// TwinCAT 3 PLC project PLC_MOTION
// Title: PLC_MOTION_LAYER
// Author: D. Hauer
// ProjectVersion: 01.00.34
// Description: MC-PtP, NCI, Camming cyclic execution layer for motion commands
// ProgramVersion: 3.1.4026.19
// libraries:
//   Tc2_EtherCAT, * (Beckhoff Automation GmbH)
//   Tc2_MC2, * (Beckhoff Automation GmbH)
//   Tc2_MC2_Camming, * (Beckhoff Automation GmbH)
//   Tc2_MC2_Drive, * (Beckhoff Automation GmbH)
//   Tc2_MC2_XFC, * (Beckhoff Automation GmbH)
//   Tc2_NCI, * (Beckhoff Automation GmbH)
//   Tc2_PlcInterpolation, * (Beckhoff Automation GmbH)
//   Tc2_Standard, * (Beckhoff Automation GmbH)
//   Tc2_System, * (Beckhoff Automation GmbH)
//   Tc2_Utilities, * (Beckhoff Automation GmbH)
//   Tc3_Module, * (Beckhoff Automation GmbH)
// project tree:
//   / CAM.TcPOU, FUNCTIONS.TcPOU, NCI.TcPOU, MAIN.TcPOU, PlcTask.TcTTO, Visualization Manager.TcVMO (not stored)
//   CAM/ FB_CamAxis.TcPOU, FB_CamCtrl.TcPOU, I_Cam_Ctrl.TcIO
//   CAM/types/ ST_CAM_CTRL.TcDUT (not stored), ST_CAM_DATA.TcDUT (not stored), ST_CAM_INFO.TcDUT (not stored), ST_CAM_READ_VALUES_PARAMETER.TcDUT, ST_CAM_STATE.TcDUT (not stored), ST_CAM_OPTIONS.TcDUT (not stored), ST_CAM_SCALING_DATA.TcDUT, ST_MOTION_FUNCTION.TcDUT (not stored), ST_MOTION_FUNCTION_POINT.TcDUT (not stored)
//   FUNCTIONS/TOUCH_PROBE/ FB_TouchProbe.TcPOU, I_TouchProbe.TcIO
//   FUNCTIONS/TOUCH_PROBE/types/ ST_2BIT.TcDUT (not stored), ST_CTRL_TOUCH_PROBE.TcDUT (not stored), ST_DC_Input.TcDUT (not stored), ST_MTI_INPUT.TcDUT (not stored), ST_MTI_STATUS.TcDUT (not stored), ST_STATE_TOUCH_PROBE.TcDUT (not stored)
//   FUNCTIONS/TRIGGER_BOX/ FB_TriggerBox.TcPOU, I_TriggerBox.TcIO
//   FUNCTIONS/TRIGGER_BOX/types/ ST_CTRL_TRIGGER.TcDUT (not stored), ST_DC_Output.TcDUT (not stored), ST_DC_State.TcDUT (not stored), ST_STATE_TRIGGER.TcDUT, T_TriggerControlBits.TcDUT
//   MAPPING/ MAPPING_in.TcPOU (not stored), MAPPING_out.TcPOU
//   MAPPING/types/ U_AXIS_CTRL.TcDUT (not stored), U_AXIS_NC_PARAMETER_WRT.TcDUT, U_AXIS_HOMING.TcDUT (not stored), U_AXIS_MOTION_OPTIONS.TcDUT, U_AXIS_MOVE_DATA.TcDUT (not stored), U_AXIS_GEAR_IN.TcDUT (not stored), U_AXIS_NC_PARAMETER_RD.TcDUT, U_AXIS_STATE.TcDUT, U_AXIS_INFO.TcDUT (not stored), U_CAM_CTRL.TcDUT, U_CAM_DATA.TcDUT (not stored), U_CAM_INFO.TcDUT (not stored), U_CAM_STATE.TcDUT (not stored), U_TOUCH_PROBE_CTRL.TcDUT (not stored), U_TOUCH_PROBE_STATE.TcDUT, U_TRIGGER_CTRL.TcDUT (not stored), U_TRIGGER_STATE.TcDUT
//   NCI/ FB_NciChannelCtrl.TcPOU (not stored), FB_NciChannel.TcPOU, I_NciChannel.TcIO (not stored), I_Nci_Ctrl.TcIO
//   NCI/types/ E_NCI_CTRL.TcDUT (not stored), E_NCI_CHANNEL_ERROR.TcDUT (not stored), E_NCI_STATE.TcDUT (not stored), E_NCI_INTERPRETER_STATE.TcDUT (not stored), ST_3D_Group.TcDUT (not stored), ST_CTRL_NCI.TcDUT (not stored), ST_NCI_M_FUNC.TcDUT (not stored), ST_Index_Group.TcDUT (not stored), ST_Interface_Group.TcDUT (not stored), ST_NciChannel_Ref.TcDUT (not stored), ST_R_Parameter.TcDUT, ST_STATE_NCI.TcDUT (not stored)
//   NC_PTP/ FB_McAxisCtrl.TcPOU, FB_McAxisBase.TcPOU, I_McAxis.TcIO (not stored)
//   NC_PTP/types/axis/ E_AxisEncoderType.TcDUT (not stored), ST_HomeParams.TcDUT (not stored)
//   NC_PTP/types/control/ E_AXIS_CTRL.TcDUT (not stored), E_AXIS_STATE.TcDUT (not stored), ST_AXIS_CTRL.TcDUT (not stored), ST_AXIS_INFO.TcDUT, ST_AXIS_STATE.TcDUT (not stored), ST_GEAR_IN.TcDUT (not stored), ST_HOMING.TcDUT (not stored), ST_MOTION_OPTIONS.TcDUT, ST_MOVE_DATA.TcDUT (not stored), ST_NC_PARAMETER.TcDUT (not stored)
//   XFC/ FB_Xfc.TcPOU
//   XFC/types/ E_XFC_CHECK.TcDUT (not stored)
//   _DUT/ E_CHECK_STATE.TcDUT (not stored), E_PROGRESS.TcDUT (not stored)
//   _GVL/ GlobalTextList.TcGTLO (not stored), GVL_AXIS.TcGVL, GVL_CAM.TcGVL (not stored), GVL_FUNCTIONS.TcGVL, GVL_MSG.TcGVL (not stored), GVL_NCI.TcGVL (not stored), PLC_CONSTANT.TcGVL (not stored), PLC_VERSION.TcGVL
//   _MSG/ fb_LocalTime.TcPOU (not stored), f_MessageSet.TcPOU, MessageData.TcPOU (not stored), T_MESSAGE_LIST.TcVIS
//   _MSG/types/ e_Device.TcDUT (not stored), E_MessageType.TcDUT (not stored), E_MESSAGE_STATE.TcDUT (not stored), e_Subdevice.TcDUT (not stored), ST_Message.TcDUT (not stored)
//   _UML/ CD_PLC_MOTION.TcCD (not stored) (excluded from build)
// real-time tasks:
//   TASK PlcTask: cycle T#10ms, priority 20, ADS port 350
//   TASK PlcTask1: cycle T#10ms, priority 21, ADS port 351
// motion (NC):
//   TASK NC-Task 1 SAF: cycle T#2ms, priority 4, ADS port 501
//   TASK NC-Task 1 SVB: cycle T#10ms, priority 8, ADS port 511
//   AXIS Axis 1 (id 1)
//     OtherSettings: AllowMotionCmdToSlave=true
//     encoder EncType=1
//     drive DrvType=5
//       Analog: TorqueSetpointScale=10, ScaleFactorActTorque=0.1
//       TimeComp: TaskDelayCycles=1
//     controller CtrType=1
//       CtrPara: PriorControlFactor=1
//         Observer: BandWidth=20
//   AXIS Axis 2 (id 2)
//     OtherSettings: AllowMotionCmdToSlave=true
//     encoder EncType=1
//     drive DrvType=5
//       Analog: TorqueSetpointScale=10, ScaleFactorActTorque=0.1
//       TimeComp: TaskDelayCycles=1
//     controller CtrType=1
//       CtrPara: PriorControlFactor=1
//         Observer: BandWidth=20
//   AXIS Axis 3 (id 3)
//     OtherSettings: AllowMotionCmdToSlave=true
//     encoder EncType=1
//     drive DrvType=5
//       Analog: TorqueSetpointScale=10, ScaleFactorActTorque=0.1
//       TimeComp: TaskDelayCycles=1
//     controller CtrType=1
//       CtrPara: PriorControlFactor=1
//         Observer: BandWidth=20
//   AXIS Axis 4 (id 4)
//     OtherSettings: AllowMotionCmdToSlave=true
//     encoder EncType=1
//     drive DrvType=5
//       Analog: TorqueSetpointScale=10, ScaleFactorActTorque=0.1
//       TimeComp: TaskDelayCycles=1
//     controller CtrType=1
//       CtrPara: PriorControlFactor=1
//         Observer: BandWidth=20
//   AXIS Axis 5 (id 5)
//     OtherSettings: AllowMotionCmdToSlave=true
//     encoder EncType=1
//     drive DrvType=5
//       Analog: TorqueSetpointScale=10, ScaleFactorActTorque=0.1
//       TimeComp: TaskDelayCycles=1
//     controller CtrType=1
//       CtrPara: PriorControlFactor=1
//         Observer: BandWidth=20
//   AXIS Axis 6 (id 6)
//     OtherSettings: AllowMotionCmdToSlave=true
//     encoder EncType=1
//     drive DrvType=5
//       Analog: TorqueSetpointScale=10, ScaleFactorActTorque=0.1
//       TimeComp: TaskDelayCycles=1
//     controller CtrType=1
//       CtrPara: PriorControlFactor=1
//         Observer: BandWidth=20
// variable links:
//   PLC_MOTION/PLC_MOTION Instance <-> NC-Task 1 SAF/Axes/Axis 1
//     PlcTask Inputs/GVL_AXIS.AxisRef[1].NcToPlc <-> Outputs/ToPlc
//     PlcTask Outputs/GVL_AXIS.AxisRef[1].PlcToNc <-> Inputs/FromPlc
//   PLC_MOTION/PLC_MOTION Instance <-> NC-Task 1 SAF/Axes/Axis 2
//     PlcTask Inputs/GVL_AXIS.AxisRef[2].NcToPlc <-> Outputs/ToPlc
//     PlcTask Outputs/GVL_AXIS.AxisRef[2].PlcToNc <-> Inputs/FromPlc
//   PLC_MOTION/PLC_MOTION Instance <-> NC-Task 1 SAF/Axes/Axis 3
//     PlcTask Inputs/GVL_AXIS.AxisRef[3].NcToPlc <-> Outputs/ToPlc
//     PlcTask Outputs/GVL_AXIS.AxisRef[3].PlcToNc <-> Inputs/FromPlc
//   PLC_MOTION/PLC_MOTION Instance <-> NC-Task 1 SAF/Axes/Axis 4
//     PlcTask Inputs/GVL_AXIS.AxisRef[4].NcToPlc <-> Outputs/ToPlc
//     PlcTask Outputs/GVL_AXIS.AxisRef[4].PlcToNc <-> Inputs/FromPlc
//   PLC_MOTION/PLC_MOTION Instance <-> NC-Task 1 SAF/Axes/Axis 5
//     PlcTask Inputs/GVL_AXIS.AxisRef[5].NcToPlc <-> Outputs/ToPlc
//     PlcTask Outputs/GVL_AXIS.AxisRef[5].PlcToNc <-> Inputs/FromPlc
//   PLC_MOTION/PLC_MOTION Instance <-> NC-Task 1 SAF/Axes/Axis 6
//     PlcTask Inputs/GVL_AXIS.AxisRef[6].NcToPlc <-> Outputs/ToPlc
//     PlcTask Outputs/GVL_AXIS.AxisRef[6].PlcToNc <-> Inputs/FromPlc

CONFIGURATION PLC_MOTION
    RESOURCE PLC ON TwinCAT3
        TASK PlcTask(INTERVAL := T#10ms, PRIORITY := 20);
        PROGRAM MAPPING_in WITH PlcTask : MAPPING_in;
        PROGRAM MAIN WITH PlcTask : MAIN;
        PROGRAM FUNCTIONS WITH PlcTask : FUNCTIONS;
        PROGRAM NCI WITH PlcTask : NCI;
        PROGRAM CAM WITH PlcTask : CAM;
        PROGRAM MAPPING_out WITH PlcTask : MAPPING_out;
    END_RESOURCE
END_CONFIGURATION

// ---- CAM/types/ST_CAM_READ_VALUES_PARAMETER.TcDUT
{attribute 'pack_mode' := '2'}
TYPE ST_CAM_READ_VALUES_PARAMETER :
STRUCT
  nValueSelectMask        : UINT;   // ReadMotionFunctionValues
  rValueMasterStart       : LREAL;  // ReadMotionFunctionValues
  rValueMasterEnd         : LREAL;  // ReadMotionFunctionValues
  rIncrement              : LREAL;
END_STRUCT
END_TYPE

// ---- CAM/types/ST_CAM_SCALING_DATA.TcDUT
{attribute 'pack_mode' := '2'}
TYPE ST_CAM_SCALING_DATA :
STRUCT
  bMasterRelative         : BIT;
  bSlaveRelative          : BIT;

  // scaling of X-axis (Master) of the CAM
  nMasterScalingMode      : UINT;
  rMasterOffset           : LREAL;
  rMasterScaling          : LREAL := 1.0;

  // scaling of Y-axis (Slave) of CAM
  nSlaveScalingMode       : UINT;

  rSlaveOffset            : LREAL;
  rSlaveScaling           : LREAL := 1.0;
END_STRUCT
END_TYPE

// ---- FUNCTIONS/TRIGGER_BOX/types/ST_STATE_TRIGGER.TcDUT
TYPE ST_STATE_TRIGGER :
STRUCT
  State           : UINT; // 0 := deactivated, 100 := BUSY, 1000 := DONE, 9000 := ERROR
  Init            : UINT;
  // FlashTimestamp  : ARRAY[1..GVL_FUNCTIONS.MAX_TRIGGER_COUNT] OF ULINT; // DC timestamp
  FlashPosition   : ARRAY[1..MAX_TRIGGER_COUNT] OF LREAL; // AxisPosition for DC timestamp
END_STRUCT
END_TYPE

// ---- FUNCTIONS/TRIGGER_BOX/types/T_TriggerControlBits.TcDUT
TYPE T_TriggerControlBits :
STRUCT
  Enable        : BIT;
  Init          : BIT;
  NoFeedback    : BIT;
{attribute 'hide'} 
  b3            : BIT;
{attribute 'hide'} 
  b4            : BIT;
{attribute 'hide'} 
  b5            : BIT;
{attribute 'hide'} 
  b6            : BIT;
{attribute 'hide'} 
  b7            : BIT;
END_STRUCT
END_TYPE

// ---- MAPPING/types/U_AXIS_NC_PARAMETER_WRT.TcDUT
TYPE U_AXIS_NC_PARAMETER_WRT :
UNION

  stCtrl              : ARRAY[1..MAX_AXIS] OF ST_NC_PARAMETER;

{IF defined (AXIS_MAP)}
  {info 'U_AXIS_NC_PARAMETER_WRT mapping activated'}
  byCtrl    AT %I*    : ARRAY[1..MAX_AXIS] OF
                        ARRAY[1..SIZEOF(ST_NC_PARAMETER)] OF BYTE;
{ELSE}
  byCtrl              : ARRAY[1..MAX_AXIS] OF
                        ARRAY[1..SIZEOF(ST_NC_PARAMETER)] OF BYTE;
{END_IF}
END_UNION
END_TYPE

// ---- MAPPING/types/U_AXIS_MOTION_OPTIONS.TcDUT
TYPE U_AXIS_MOTION_OPTIONS :
UNION

  stCtrl              : ARRAY[1..MAX_AXIS] OF ST_MOTION_OPTIONS;

{IF defined (AXIS_MAP)}
  {info 'U_AXIS_MOTION_OPTIONS mapping activated'}
  byCtrl    AT %I*    : ARRAY[1..MAX_AXIS] OF
                        ARRAY[1..SIZEOF(ST_MOTION_OPTIONS)] OF BYTE;
{ELSE}
  byCtrl              : ARRAY[1..MAX_AXIS] OF
                        ARRAY[1..SIZEOF(ST_MOTION_OPTIONS)] OF BYTE;
{END_IF}
END_UNION
END_TYPE

// ---- MAPPING/types/U_AXIS_NC_PARAMETER_RD.TcDUT
TYPE U_AXIS_NC_PARAMETER_RD :
UNION

  stState             : ARRAY[1..MAX_AXIS] OF ST_NC_PARAMETER;

{IF defined (AXIS_MAP)}
  {info 'U_AXIS_NC_PARAMETER_RD mapping activated'}
  byState   AT %Q*    : ARRAY[1..MAX_AXIS] OF
                        ARRAY[1..SIZEOF(ST_NC_PARAMETER)] OF BYTE;
{ELSE}
  byState             : ARRAY[1..MAX_AXIS] OF
                        ARRAY[1..SIZEOF(ST_NC_PARAMETER)] OF BYTE;
{END_IF}
END_UNION
END_TYPE

// ---- MAPPING/types/U_AXIS_STATE.TcDUT
TYPE U_AXIS_STATE :
UNION

  stState             : ARRAY[1..MAX_AXIS] OF ST_AXIS_STATE;

{IF defined (AXIS_MAP)}
  {info 'U_AXIS_STATE mapping activated'}
  byState   AT %Q*    : ARRAY[1..MAX_AXIS] OF
                        ARRAY[1..SIZEOF(ST_AXIS_STATE)] OF BYTE;
{ELSE}
  byState             : ARRAY[1..MAX_AXIS] OF
                        ARRAY[1..SIZEOF(ST_AXIS_STATE)] OF BYTE;
{END_IF}
END_UNION
END_TYPE

// ---- MAPPING/types/U_CAM_CTRL.TcDUT
TYPE U_CAM_CTRL :
UNION
  stCtrl              : ARRAY[1..MAX_AXIS] OF ST_CAM_CTRL;

{IF defined (CAM_MAP)}
  {info 'U_CAM_CTRL mapping activated'}
  byCtrl    AT %I*    : ARRAY[1..MAX_AXIS] OF
                        ARRAY[1..SIZEOF(ST_CAM_CTRL)] OF BYTE;
{ELSE}
  byCtrl              : ARRAY[1..MAX_AXIS] OF
                        ARRAY[1..SIZEOF(ST_CAM_CTRL)] OF BYTE;
{END_IF}
END_UNION
END_TYPE

// ---- MAPPING/types/U_TOUCH_PROBE_STATE.TcDUT
TYPE U_TOUCH_PROBE_STATE :
UNION
  stState              : ARRAY[1..MAX_TOUCH_PROBE] OF ST_STATE_TOUCH_PROBE;

{IF defined (TRIGGER_MAP)}
  {info 'U_TOUCH_PROBE_STATE mapping activated'}
  byState    AT %Q*   : ARRAY[1..MAX_TOUCH_PROBE] OF
                        ARRAY[1..SIZEOF(ST_STATE_TOUCH_PROBE)] OF BYTE;
{ELSE}
  byState             : ARRAY[1..MAX_TOUCH_PROBE] OF
                        ARRAY[1..SIZEOF(ST_STATE_TOUCH_PROBE)] OF BYTE;
{END_IF}
END_UNION
END_TYPE

// ---- MAPPING/types/U_TRIGGER_STATE.TcDUT
TYPE U_TRIGGER_STATE :
UNION
  stState              : ARRAY[1..MAX_TRIGGER_BOX] OF ST_STATE_TRIGGER;

{IF defined (TRIGGER_MAP)}
  {info 'U_TRIGGER_STATE mapping activated'}
  byState    AT %Q*   : ARRAY[1..MAX_TRIGGER_BOX] OF
                        ARRAY[1..SIZEOF(ST_STATE_TRIGGER)] OF BYTE;
{ELSE}
  byState             : ARRAY[1..MAX_TRIGGER_BOX] OF
                        ARRAY[1..SIZEOF(ST_STATE_TRIGGER)] OF BYTE;
{END_IF}
END_UNION
END_TYPE

// ---- NCI/types/ST_R_Parameter.TcDUT
{attribute 'pack_mode' := '2'}
TYPE ST_R_Parameter :
STRUCT
  _nStart               : DINT := 901;
  _nCount               : DINT :=   4;
  _rValue               : ARRAY[0..MAX_R_PARA] OF LREAL;
END_STRUCT
END_TYPE

// ---- NC_PTP/types/control/ST_AXIS_INFO.TcDUT
{attribute 'pack_mode' := '2'}
TYPE ST_AXIS_INFO :
STRUCT
  bEnabled    : BIT; // Enabled: check if ControlLoop is closed and active
  bReferenced : BIT; // Axis homing bit
  bReady      : BIT; // enabled & NOT bError & no Axis Function requested
  bBusy       : BIT; // axis function requested or active
  bError      : BIT;
  bTimeout    : BIT; // for move cmds or switching drive on timeout
  bInTarget   : BIT; // ActPos = SetPos --> position check is done with configured window in NC
  bStandstill : BIT; // No Error and NOT moving
 
  nErrorId            : UDINT;

  rActPos             : LREAL;
  rActVelo            : LREAL;
  rPosDiff            : LREAL;

  dwCoupleState       : DWORD;   // cyclic information about axis couple state
  nNcAxisId           : UDINT;
END_STRUCT
END_TYPE

// ---- NC_PTP/types/control/ST_MOTION_OPTIONS.TcDUT
{attribute 'pack_mode' := '2'}
TYPE ST_MOTION_OPTIONS :
STRUCT
  eBufferMode   : Tc2_MC2.MC_BufferMode;  // used in FB_McAxisCtrl.MoverBufferPos, MoveBufferVelo
  rDistance     : LREAL;                  // used in FB_McAxis.SendToPos; axis has to move rDistance for method to be done
END_STRUCT
END_TYPE

// ---- _GVL/GVL_AXIS.TcGVL
{attribute 'qualified_only'}
VAR_GLOBAL

  // TwinCAT NC mapping cyclic reference
  //  - link to NC/PtP
  //  - a motion Ctrl function block gets REFERENCE TO all axis
  AxisRef                     : ARRAY[1..PLC_CONSTANT.MAX_AXIS] OF Tc2_MC2.AXIS_REF;

  //-----------------------------------------------------------------------------
  // interfaces of I_McAxis 
  //  - to provide access to basic MC functions in 
  //    - NCI(PRG)() / FB_NciChannelCtrl,
  //    - CAM(PRG)() / FB_CamCtrl
  //-----------------------------------------------------------------------------
  ItfMcAxis                   : ARRAY[1..PLC_CONSTANT.MAX_AXIS] OF I_McAxis;     // interface to basic MC functions


  //-----------------------------------------------------------------------------
  // command and state structure
  //  - datafields for anyone to access
  //    - ADS via symbol
  //    - cyclic mapping to any other cyclic network/runtime
  //-----------------------------------------------------------------------------
  Ctrl                        : ARRAY[1..PLC_CONSTANT.MAX_AXIS] OF ST_AXIS_CTRL;      // command structure to write into
  State                       : ARRAY[1..PLC_CONSTANT.MAX_AXIS] OF ST_AXIS_STATE;     // state structure to read from

  //-----------------------------------------------------------------------------
  // data and info structure
  //  - parameter data fields for
  //    - Ctrl  --> Data
  //    - State --> Info
  //-----------------------------------------------------------------------------
  Info                        : ARRAY[1..PLC_CONSTANT.MAX_AXIS] OF ST_AXIS_INFO;      // axis state and position data to read from
  Data                        : ARRAY[1..PLC_CONSTANT.MAX_AXIS] OF ST_MOVE_DATA;      // axis data to write into


  //-----------------------------------------------------------------------------
  // special function parameter structs
  // - additional details for axis command
  //-----------------------------------------------------------------------------
  NcParameterWrt              : ARRAY[1..PLC_CONSTANT.MAX_AXIS] OF ST_NC_PARAMETER;   // struct for a single parameter value put/get your data here before/after using Ctrl
  NcParameterRd               : ARRAY[1..PLC_CONSTANT.MAX_AXIS] OF ST_NC_PARAMETER;   // struct for a single parameter value put/get your data here before/after using Ctrl

  HomeParameter               : ARRAY[1..PLC_CONSTANT.MAX_AXIS] OF ST_HOMING;         // homing parameter for each axis

  GearInParameter             : ARRAY[1..PLC_CONSTANT.MAX_AXIS] OF ST_GEAR_IN;        // GearIn and GearInMultiMaster, index to master axes[1-4], rGearRatio[1-4]

  MotionOptions               : ARRAY[1..PLC_CONSTANT.MAX_AXIS] OF ST_MOTION_OPTIONS; // additional motion parameters


  //-----------------------------------------------------------------------------
  // cyclic interface function block: FB_McAxisCtrl
  //  - PtP MC functions are here
  //  - implements I_McAxis
  //-----------------------------------------------------------------------------
  Control                     : ARRAY[1..PLC_CONSTANT.MAX_AXIS] OF FB_McAxisCtrl;     // cyclic interface for accepting and executing orders

END_VAR

// ---- _GVL/GVL_FUNCTIONS.TcGVL
{attribute 'qualified_only'}
VAR_GLOBAL
  //-----------------------------------------------------------------------------------------------------------
  // TriggerBox for moving axis, set output to activate camera, get input timestamp from flash controller
  //-----------------------------------------------------------------------------------------------------------
{IF defined (XFC)}
  TriggerBoxCtrl                : ARRAY[1..MAX_TRIGGER_BOX] OF Fb_TriggerBox;   // execution of trigger function
{ELSE}
  TriggerBoxCtrl                : ARRAY[1..MAX_TRIGGER_BOX] OF I_TriggerBox;   // execution of trigger function
{END_IF}

  CtrlTrigger                   : ARRAY[1..MAX_TRIGGER_BOX] OF ST_CTRL_TRIGGER;
  StateTrigger                  : ARRAY[1..MAX_TRIGGER_BOX] OF ST_STATE_TRIGGER;

  DigitalOutPutDCState  AT %I*  : ARRAY[1..MAX_TRIGGER_BOX] OF ST_DC_State;

  DigitalOutputDC   AT %Q*      : ARRAY[1..MAX_TRIGGER_BOX] OF ST_DC_Output;
  DigitalInputDC    AT %I*      : ARRAY[1..MAX_TRIGGER_BOX] OF ST_DC_Input; // distributed clock digital input with timestamps positive & negative


  //-----------------------------------------------------------------------------------------------------------
  // Touch Probe with moving axis, get input timestamp within axis window, get prcise position using the timestamp
  //-----------------------------------------------------------------------------------------------------------
{IF defined (XFC)}
  TouchProbeCtrl                : ARRAY[1..MAX_TOUCH_PROBE] OF Fb_TouchProbe;   // execution of Touch probe function
{ELSE}
  TouchProbeCtrl                : ARRAY[1..MAX_TOUCH_PROBE] OF I_TouchProbe;   // execution of Touch probe function
{END_IF}

  CtrlTouchProbe                : ARRAY[1..MAX_TOUCH_PROBE] OF ST_CTRL_TOUCH_PROBE;
  StateTouchProbe               : ARRAY[1..MAX_TOUCH_PROBE] OF ST_STATE_TOUCH_PROBE;

  //DigitalInputDC    AT %I*      : ARRAY[1..MAX_TOUCH_PROBE] OF ST_DC_Input; // distributed clock digital input with timestamps positive & negative
  DigitalInput      AT %I*      : ARRAY[1..MAX_TOUCH_PROBE] OF ST_MTI_INPUT;    // multi time stamp, one channel
  DigitalState      AT %I*      : ARRAY[1..MAX_TOUCH_PROBE] OF ST_MTI_STATUS;   // multi time stamp status from terminal

END_VAR

// ---- _GVL/PLC_VERSION.TcGVL
{attribute 'qualified_only'}
VAR_GLOBAL CONSTANT
  VERSION               : STRING := 'V 01.00.34';

  // 2025 10 24 HAUD
  //
  // documentation added, 
  // project dev changed to 4026.19
  // Ambiguities resoved

  // 2025 08 21 HAUD
  //
  // e_Device: Application added
  // e_Subdevices: merge with XTS_TRANSPORT_LAYER
  // FB_McAxis: testing SendToPos, distance added to method interface

  // 2025 02 17 HAUD
  //
  // code review
  // Message Levels are set during initialization
  // sizeof mapping data is fetched at startup only

  // 2025 01 09 HAUD
  //
  // - FUNCTIONS
  //    - code review
  //    - ctrl/state mechanic harmonized
  // - MAPPING
  //    - UNIONS added

  // 2024 08 08 HAUD
  //
  // - TC_PLC_MOTION_LAYER: 
  //    - XFC base class added
  //    - TriggerBox (DC output set, DC Input latch)
  //    - TouchProbe (DC Input latch: positive, negative)

  // 2024 06 21 HAUD
  //
  // - TC_PLC_MOTION_LAYER: 
  //    - E_PROGRESS refactoring to match TC_XTS_TRANSPORT_LAYER
  

  // 2024 06 10 HAUD
  //
  // - TC_PLC_MOTION_LAYER: 
  //    - rename repository
  //    - remove LEGACY compatibility
  //
  // - PLC_OPEN_DRIVE:
  //    - deprecated


  // 2024 05 31 HAUD
  // 
  // V 01.00.02
  // precompiler defines: 
  //  - BSD: 
  //    - Tc-BSD file system is used else Windows file system is used
  //
  //  - TEST:
  //    - GVL_MSG.MessageLevel
  // Axis, Cam, Nci have individual message levels now

  // 2024 03 09 HAUD
  // 
  // V 01.00.01
  // MC PtP - execution layer with optional mapping
  // NCI    - execution layer with optional mapping
  // CAM    . execution layer with optional mapping
  // precompiler defines: 
  //  - WIN: windows file system is used else Tc-BSD file system is used
  //  - NCI: NCI libraries are linked in project
  //  - CAM: Camming libraries are linked in project
  //  - AXIS_MAP: mapping is used


  // 2024 02 15 HAUD
  // 
  // V 00.50.04
  //
  // Buffered moves test
  // CamIn Test --> TODO MultiCam
  // Message system, cyclic check for write
  

  // 2024 01 12 HAUD
  //
  // V 00.50.03
  //
  // Building is done
  // start of UnitTesting

  // 2024 01 17 HAUD
  //
  // V 00.50.02
  // 
  // start camming implementation (MC_CamIn_V2)
  // legacy namespace available for downward compatibility of ADS Symbol names

  // 2023 12 23 HAUD
  // NC_PTP
  // - redesign for PLC_OPEN_DRIVE started 
  //    --> E_PROGRESS for state feedback
  // - FB_AxisControl inherits FB_McAxis


  //  2023 10 19
  //  HAUD
  // first draft 
  // TODO: everything

END_VAR

// ---- CAM/I_Cam_Ctrl.TcIO
INTERFACE I_Cam_Ctrl

PROPERTY Axes : reference TO ARRAY[1..PLC_CONSTANT.MAX_AXIS] OF AXIS_REF
SET
END_SET
END_PROPERTY

PROPERTY AxisCtrl : pointer to ARRAY[1..PLC_CONSTANT.MAX_AXIS] OF st_axis_ctrl
SET
END_SET
END_PROPERTY

PROPERTY AxisData : pointer to ARRAY[1..PLC_CONSTANT.MAX_AXIS] OF ST_CAM_DATA
SET
END_SET
END_PROPERTY

PROPERTY AxisIndex : uint
SET
END_SET
END_PROPERTY

PROPERTY AxisInfo : pointer to ARRAY[1..PLC_CONSTANT.MAX_AXIS] OF ST_AXIS_INFO
SET
END_SET
END_PROPERTY

PROPERTY AxisState : pointer to ARRAY[1..PLC_CONSTANT.MAX_AXIS] OF ST_CAM_STATE
SET
END_SET
END_PROPERTY

METHOD Cycle  : e_progress
END_METHOD

PROPERTY ItfMcAxes : array[1..MAX_AXIS] of I_McAxis
SET
END_SET
END_PROPERTY

PROPERTY MessageLevel : E_MessageType
SET
END_SET
END_PROPERTY

PROPERTY MotionFunction : POINTER TO ARRAY[1..MAX_AXIS] OF ST_MOTION_FUNCTION
SET
END_SET
END_PROPERTY

PROPERTY MotionFunctionPoint : pointer to array[1..MAX_AXIS] of ST_MOTION_FUNCTION_POINT
SET
END_SET
END_PROPERTY

END_INTERFACE

// ---- FUNCTIONS/TOUCH_PROBE/I_TouchProbe.TcIO
INTERFACE I_TouchProbe

PROPERTY Ctrl : REFERENCE TO ARRAY [1..MAX_TOUCH_PROBE] OF ST_CTRL_TOUCH_PROBE
SET
END_SET
END_PROPERTY

METHOD Cycle : BOOL
VAR_INPUT
END_VAR
END_METHOD

PROPERTY Index : udint
GET
END_GET
SET
END_SET
END_PROPERTY

PROPERTY Input : pointer TO ARRAY [1..MAX_TOUCH_PROBE] OF ST_MTI_Input
SET
END_SET
END_PROPERTY

PROPERTY InputState : pointer TO ARRAY [1..MAX_TOUCH_PROBE] OF ST_MTI_STATUS
SET
END_SET
END_PROPERTY

PROPERTY ItfAxis : ARRAY[1..MAX_AXIS]       OF I_McAxis
SET
END_SET
END_PROPERTY

PROPERTY MessageLevel : e_messagetype
GET
END_GET
SET
END_SET
END_PROPERTY

PROPERTY State :  REFERENCE TO ARRAY[1..MAX_TOUCH_PROBE] OF ST_STATE_TOUCH_PROBE;
SET
END_SET
END_PROPERTY

END_INTERFACE

// ---- FUNCTIONS/TRIGGER_BOX/I_TriggerBox.TcIO
INTERFACE I_TriggerBox

PROPERTY Ctrl : REFERENCE TO ARRAY [1..MAX_TRIGGER_BOX] OF ST_CTRL_TRIGGER
SET
END_SET
END_PROPERTY

METHOD Cycle : BOOL
VAR_INPUT
END_VAR
END_METHOD

METHOD CycleWaitForPosition : BOOL
VAR_INPUT
END_VAR
END_METHOD

PROPERTY Index : udint
GET
END_GET
SET
END_SET
END_PROPERTY

PROPERTY Input : pointer TO ARRAY [1..MAX_TRIGGER_BOX] OF ST_DC_Input
SET
END_SET
END_PROPERTY

PROPERTY ItfAxis : ARRAY[1..MAX_AXIS]       OF I_McAxis
SET
END_SET
END_PROPERTY

PROPERTY MessageLevel : e_messagetype
GET
END_GET
SET
END_SET
END_PROPERTY

PROPERTY Output_2252 : pointer TO ARRAY [1..MAX_TRIGGER_BOX] OF ST_DC_Output
SET
END_SET
END_PROPERTY

PROPERTY State : REFERENCE TO ARRAY[1..MAX_TRIGGER_BOX] OF ST_STATE_TRIGGER
SET
END_SET
END_PROPERTY

END_INTERFACE

// ---- NCI/I_Nci_Ctrl.TcIO
INTERFACE I_Nci_Ctrl

PROPERTY ChnCtrl : pointer to ST_CTRL_NCI
SET
END_SET
END_PROPERTY

PROPERTY ChnId : udint
GET
END_GET
END_PROPERTY

PROPERTY ChnState : pointer to ST_STATE_NCI
SET
END_SET
END_PROPERTY

METHOD Cycle : E_PROGRESS
VAR_INPUT
END_VAR
END_METHOD

PROPERTY ItfChannel : I_NciChannel
GET
END_GET
END_PROPERTY

PROPERTY M_FunctionScope : pointer to st_nci_m_func
SET
END_SET
END_PROPERTY

END_INTERFACE

// ---- MAIN.TcPOU
PROGRAM MAIN
VAR
  bInit                     : BOOL;         // shall be checked by controlling entity, before using Ctrl/State structs
  eInit                     : E_PROGRESS;   // shall be checked by controlling entity, before using Ctrl/State structs

  nAxis,
  nAxisInit                 : UINT;

  stMsg                     : ST_Message;

  bWriteTimerActive         : Bool;         // you decide whether to use timed logging into file or not
  tWriteLog                 : TIME := T#10S;
  tonWriteLog               : Tc2_Standard.TON;
END_VAR


(*
//-----------------------------------------------------------------------------------------------------------------
//-----------------------------------------------------------------------------------------------------------------
// react to operation modes (how to do it in an easy self documenting way)
//-----------------------------------------------------------------------------------------------------------------
//-----------------------------------------------------------------------------------------------------------------
CASE (GVL_AXIS.State[i].eState MOD E_PROGRESS.PROGRESS_DONE)
OF
  E_AXIS_STATE.AXIS_INIT:
    ;// do something after success  

  E_AXIS_STATE.AXIS_MOVE_POS::
    ;// do something after success
ELSE
  CASE (GVL_AXIS.State[i].eState MOD E_PROGRESS.PROGRESS_ERROR)
  OF
    E_AXIS_STATE.AXIS_INIT:
      ;// do something after success  
  
    E_AXIS_STATE.AXIS_MOVE_POS::
      ;// do something after success
  ELSE
    ;// down the rabbit hole you go from here
  END_CASE
END_CASE
*)



//-----------------------------------------------------------------------------------------------------------------
// Local time; used for timestamps
//-----------------------------------------------------------------------------------------------------------------
GVL_MSG.fbLocalTime(
                    sLocalTime                => GVL_MSG.sLocalTime, 
                    dtLocalTime               => GVL_MSG.dtLocalTime);
//-----------------------------------------------------------------------------------------------------------------
//-----------------------------------------------------------------------------------------------------------------
// /assign dataflow
//-----------------------------------------------------------------------------------------------------------------
FOR nAxis := 1 TO PLC_CONSTANT.MAX_AXIS
DO
  GVL_AXIS.Control[nAxis].AxisIndex           := nAxis;

  GVL_AXIS.Control[nAxis].AxisCtrl            := ADR(GVL_AXIS.Ctrl);          // command
  GVL_AXIS.Control[nAxis].AxisState           := ADR(GVL_AXIS.State);         // state + result of command

  GVL_AXIS.Control[nAxis].Axes                REF=   GVL_AXIS.AxisRef;        // All for one; coupling requires access across all axes

  GVL_AXIS.Control[nAxis].AxisInfo            := ADR(GVL_AXIS.Info);          // axis information: act/set values and bits from axis
  GVL_AXIS.Control[nAxis].AxisData            := ADR(GVL_AXIS.Data);          // position and dynamic constraints for movement
  GVL_AXIS.Control[nAxis].AxisGearInParameter := ADR(GVL_AXIS.GearInParameter);

  GVL_AXIS.Control[nAxis].WriteNcParameter    := ADR(GVL_AXIS.NcParameterWrt);
  GVL_AXIS.Control[nAxis].ReadNcParameter     := ADR(GVL_AXIS.NcParameterRd);

  GVL_AXIS.Control[nAxis].HomingParameter     := ADR(GVL_AXIS.HomeParameter);
  GVL_AXIS.Control[nAxis].MotionOptions       := ADR(GVL_AXIS.MotionOptions);

  GVL_AXIS.ItfMcAxis[nAxis]                   := GVL_AXIS.Control[nAxis]; 
END_FOR
//-----------------------------------------------------------------------------------------------------------------
// assign dataflow/
//-----------------------------------------------------------------------------------------------------------------
//-----------------------------------------------------------------------------------------------------------------
// /INIT
// - successful init is required for other optional members to start
//-----------------------------------------------------------------------------------------------------------------
IF NOT bInit
THEN
  CASE eInit
  OF
    E_PROGRESS.PROGRESS_INVALID,
    E_PROGRESS.PROGRESS_DONE:
      FOR nAxis := 1 TO PLC_CONSTANT.MAX_AXIS
      DO
        GVL_AXIS.Control[nAxis].MessageLevel  := GVL_MSG.MessageLevelAxisPtp;
      END_FOR
      nAxisInit                               := 1;
      eInit                                   := E_PROGRESS.PROGRESS_INIT;


    E_PROGRESS.PROGRESS_INIT:
      stMsg.eType                             := E_MessageType.eMessageVerbose;
      stMsg.eDevice                           := e_Device.General;
      stMsg.eSubdevice                        := e_SubDevice.AxisStartUp;
      stMsg.iErrorNumber                      := nAxisInit;

      stMsg.sText                             := concat('MAIN.eInit: ', TO_STRING(eInit));

      IF (GVL_MSG.MessageLevelAxisPtp = E_MessageType.eMessageVerbose)
      THEN
        f_MessageSet(stMsg);
      END_IF

      GVL_AXIS.Ctrl[nAxisInit].eCmd           := E_AXIS_CTRL.AXIS_NULL;
      eInit                                   := E_PROGRESS.PROGRESS_BUSY;


    E_PROGRESS.PROGRESS_BUSY:
      GVL_AXIS.Ctrl[nAxisInit].eCmd          := E_AXIS_CTRL.AXIS_INIT;

      IF    (GVL_AXIS.State[nAxisInit].eState = E_AXIS_STATE.AXIS_INIT + E_PROGRESS.PROGRESS_ERROR)
      THEN
        eInit                                 := E_PROGRESS.PROGRESS_ERROR;

        stMsg.eType                           := E_MessageType.eMessageError;
        stMsg.eDevice                         := e_Device.General;
        stMsg.eSubdevice                      := e_SubDevice.AxisStartUp;
        stMsg.iErrorNumber                    := GVL_AXIS.Control[nAxisInit].ErrorId;

        stMsg.sText                           := concat('MAIN.eInit ERROR at Index: ', TO_STRING(nAxisInit));
        f_MessageSet(stMsg);

      ELSIF (GVL_AXIS.State[nAxisInit].eState = E_AXIS_STATE.AXIS_INIT + E_PROGRESS.PROGRESS_DONE)
      THEN
        eInit                                 := E_PROGRESS.PROGRESS_CHECK;
      END_IF


    E_PROGRESS.PROGRESS_CHECK:
      IF NOT (nAxisInit > PLC_CONSTANT.MAX_AXIS-1)
      THEN
        nAxisInit                             := nAxisInit + 1;
        eInit                                 := E_PROGRESS.PROGRESS_INIT;

      ELSE
        bInit                                 := TRUE;
        eInit                                 := E_PROGRESS.PROGRESS_DONE;

        stMsg.eType                           := E_MessageType.eMessageInfo;
        stMsg.eDevice                         := e_Device.General;
        stMsg.eSubdevice                      := e_SubDevice.AxisStartUp;
        stMsg.iErrorNumber                    := MAX_AXIS;

        stMsg.sText                           := concat('MAIN.eInit: ', TO_STRING(eInit));
        f_MessageSet(stMsg);
      END_IF
  END_CASE
END_IF
//-----------------------------------------------------------------------------------------------------------------
// INIT
//-----------------------------------------------------------------------------------------------------------------
//-----------------------------------------------------------------------------------------------------------------
// /cyclic
//-----------------------------------------------------------------------------------------------------------------
IF (eInit <> E_PROGRESS.PROGRESS_ERROR)
THEN
  FOR nAxis := 1 TO PLC_CONSTANT.MAX_AXIS
  DO
      GVL_AXIS.Control[nAxis]();
  END_FOR
END_IF
//-----------------------------------------------------------------------------------------------------------------
// cyclic/
//-----------------------------------------------------------------------------------------------------------------


//-----------------------------------------------------------------------------------------------------------------
// /logging
//-----------------------------------------------------------------------------------------------------------------
tonWriteLog(IN:= TRUE, PT := tWriteLog);

IF (tonWriteLog.Q)
THEN
  MessageData.bWriteFile      := bWriteTimerActive; // you have to decide whether to use timed write or not
  tonWriteLog(IN:= FALSE);
END_IF

//-----------------------------------------------------------------------------------------------------------------
// write message list to file
//-----------------------------------------------------------------------------------------------------------------
MessageData(pList			        := ADR(GVL_MSG.Messages),
			      pLocalTime        := ADR(GVL_MSG.dtLocalTime), 
			      bBusy=> );

// clear write trigger
IF MessageData.bWriteFile AND
   MessageData.bBusy
THEN
  MessageData.bWriteFile      := FALSE;
END_IF
//-----------------------------------------------------------------------------------------------------------------
// logging/
//-----------------------------------------------------------------------------------------------------------------

END_PROGRAM

// ---- _MSG/f_MessageSet.TcPOU
FUNCTION f_MessageSet : BOOL
VAR_INPUT
  stMessage   : ST_Message;
END_VAR
VAR
  _uiIndex   : uINT;
END_VAR

stMessage.tTime                     := GVL_MSG.sLocalTime;

FOR _uiIndex := 1 TO GVL_MSG.MAX_MESSAGE
DO
  IF (GVL_MSG.Messages[_uiIndex].eType = e_MessageType.eMessageEmpty)
  THEN
    GVL_MSG.Messages[_uiIndex]      := stMessage;
    GVL_MSG.MessageIndex            := _uiIndex;
    EXIT;
  END_IF
END_FOR

IF (stMessage.eType = E_MessageType.eMessageError)
THEN
  // in case of error: increment counter
  GVL_MSG.MessageError := GVL_MSG.MessageError + 1;
END_IF

END_FUNCTION

// ---- FUNCTIONS.TcPOU
PROGRAM FUNCTIONS
VAR
  eInit             : E_PROGRESS;

  nAxis,
  nTrigger,
  nProbe            : UINT;
END_VAR

//-----------------------------------------------------------------------------------------------------------------
// check if compiler define is present [PLC_STATE_DRIVE/CompilerDefines/Manual: XFC]
// see PLC_CONSTANT for conditional pragma
//-----------------------------------------------------------------------------------------------------------------
IF NOT PLC_CONSTANT.XFC_ACTIVE THEN eInit := E_PROGRESS.PROGRESS_NOT_EXIST; RETURN; END_IF
//-----------------------------------------------------------------------------------------------------------------
//-----------------------------------------------------------------------------------------------------------------
// check MAIN.eInit
//-----------------------------------------------------------------------------------------------------------------
IF NOT (MAIN.eInit = E_PROGRESS.PROGRESS_DONE) 
THEN
  // wait for MAIN to be fully initialized
  eInit                                               := E_PROGRESS.PROGRESS_INVALID; 
  RETURN; 
ELSE
  // at the moment FUNCTIONS does not require a general init procedure
  eInit                                               := E_PROGRESS.PROGRESS_DONE;    // general init done
END_IF
//-----------------------------------------------------------------------------------------------------------------
//-----------------------------------------------------------------------------------------------------------------
// /cyclic
//-----------------------------------------------------------------------------------------------------------------
FOR nProbe := 1 TO MAX_TOUCH_PROBE
DO
  GVL_FUNCTIONS.TouchProbeCtrl[nProbe].MessageLevel   := GVL_MSG.MessageLevelTouchProbe[nProbe];
  GVL_FUNCTIONS.TouchProbeCtrl[nProbe].Index          := nProbe;
  GVL_FUNCTIONS.TouchProbeCtrl[nProbe].ItfAxis        := GVL_AXIS.ItfMcAxis;

  GVL_FUNCTIONS.TouchProbeCtrl[nProbe].Ctrl           REF= GVL_FUNCTIONS.CtrlTouchProbe;
  GVL_FUNCTIONS.TouchProbeCtrl[nProbe].State          REF= GVL_FUNCTIONS.StateTouchProbe;

  GVL_FUNCTIONS.TouchProbeCtrl[nProbe].Input          := ADR(GVL_FUNCTIONS.DigitalInput);
  GVL_FUNCTIONS.TouchProbeCtrl[nProbe].InputState     := ADR(GVL_FUNCTIONS.DigitalState);
  GVL_FUNCTIONS.TouchProbeCtrl[nProbe].Cycle();

END_FOR

FOR nTrigger := 1 TO MAX_TRIGGER_BOX
DO
  GVL_FUNCTIONS.TriggerBoxCtrl[nTrigger].MessageLevel := GVL_MSG.MessageLevelTriggerBox[nTrigger];
  GVL_FUNCTIONS.TriggerBoxCtrl[nTrigger].Index        := nTrigger;
  GVL_FUNCTIONS.TriggerBoxCtrl[nTrigger].ItfAxis      := GVL_AXIS.ItfMcAxis;

  GVL_FUNCTIONS.TriggerBoxCtrl[nTrigger].Ctrl         REF= GVL_FUNCTIONS.CtrlTrigger;
  GVL_FUNCTIONS.TriggerBoxCtrl[nTrigger].State        REF= GVL_FUNCTIONS.StateTrigger;

  GVL_FUNCTIONS.TriggerBoxCtrl[nTrigger].Input        := ADR(GVL_FUNCTIONS.DigitalInputDC);
  GVL_FUNCTIONS.TriggerBoxCtrl[nTrigger].Output_2252  := ADR(GVL_FUNCTIONS.DigitalOutputDC);

  GVL_FUNCTIONS.TriggerBoxCtrl[nTrigger].Cycle();
END_FOR
//-----------------------------------------------------------------------------------------------------------------
// cyclic/
//-----------------------------------------------------------------------------------------------------------------
//-----------------------------------------------------------------------------------------------------------------

END_PROGRAM

// ---- NCI.TcPOU
PROGRAM NCI
VAR
  bInit                     : BOOL;
  eInit                     : E_PROGRESS;

  nChn,
  nChnInit,
  nAxis,
  nAxisInit                 : UINT;

  stMsg                     : ST_Message;

END_VAR

//-----------------------------------------------------------------------------------------------------------------
// check if compiler define is present [PLC_STATE_DRIVE/CompilerDefines/Manual: NCI]
// see PLC_CONSTANT for conditional pragma
//-----------------------------------------------------------------------------------------------------------------
IF NOT PLC_CONSTANT.NCI_ACTIVE THEN eInit   := E_PROGRESS.PROGRESS_NOT_EXIST; RETURN; END_IF
//-----------------------------------------------------------------------------------------------------------------
//-----------------------------------------------------------------------------------------------------------------
// check for MAIN.eInit
//-----------------------------------------------------------------------------------------------------------------
IF NOT (MAIN.eInit = E_PROGRESS.PROGRESS_DONE) THEN eInit   := E_PROGRESS.PROGRESS_INVALID; RETURN; END_IF
//-----------------------------------------------------------------------------------------------------------------
//-----------------------------------------------------------------------------------------------------------------
// /assign dataflow
//-----------------------------------------------------------------------------------------------------------------
FOR nChn := 1 TO MAX_NCI_CH
DO
  // NCI axis configuration --> NC AxisId used
  GVL_NCI.fbNciCtrl[nChn].ItfChannel.CfgAxes          := ADR(GVL_NCI.stAxisConfig[nChn]);

  // R Parameter properties
  GVL_NCI.fbNciCtrl[nChn].ItfChannel.R_ParameterRead  := ADR(GVL_NCI.R_ParameterRead[nChn]);
  GVL_NCI.fbNciCtrl[nChn].ItfChannel.R_ParameterWrite := ADR(GVL_NCI.R_ParameterWrite[nChn]);

  // ProgName for channel
  GVL_NCI.fbNciCtrl[nChn].ItfChannel.Prog             := GVL_NCI.sProgName[nChn];

  // check REAL value to avoid exception
  IF NOT IsFinite(F_Real(GVL_NCI.stChannelCtrl[nChn].rOverride))
  THEN
    GVL_NCI.fbNciCtrl[nChn].ItfChannel.Override       := 0.0;
  ELSE
    GVL_NCI.fbNciCtrl[nChn].ItfChannel.Override       := GVL_NCI.stChannelCtrl[nChn].rOverride;
  END_IF

  // command and state structure assignement
  GVL_NCI.fbNciCtrl[nChn].ChnCtrl                     := ADR(GVL_NCI.stChannelCtrl[nChn]);
  GVL_NCI.fbNciCtrl[nChn].ChnState                    := ADR(GVL_NCI.stChannelState[nChn]);
END_FOR
//-----------------------------------------------------------------------------------------------------------------
// assign dataflow/
//-----------------------------------------------------------------------------------------------------------------
//-----------------------------------------------------------------------------------------------------------------
// /INIT
//-----------------------------------------------------------------------------------------------------------------
IF NOT bInit
THEN
  CASE eInit
  OF
    E_PROGRESS.PROGRESS_INVALID,
    E_PROGRESS.PROGRESS_DONE:
      FOR nChn := 1 TO MAX_NCI_CH
      DO
        GVL_NCI.fbNciCtrl[nChn].ItfChannel.MessageLevel     := GVL_MSG.MessageLevelNciChn;
      END_FOR
      nChnInit                                    := 1;
      eInit                                       := E_PROGRESS.PROGRESS_INIT;


    E_PROGRESS.PROGRESS_INIT:
      stMsg.eType                                 := E_MessageType.eMessageVerbose;
      stMsg.eDevice                               := e_Device.NciChannelCtrl;
      stMsg.eSubdevice                            := e_SubDevice.NciStartUp;
      stMsg.iErrorNumber                          := nChnInit;

      stMsg.sText                                 := concat('NCI.eInit: ', TO_STRING(eInit));
      f_MessageSet(stMsg);

      GVL_NCI.stChannelCtrl[nChnInit].eCmd        := E_NCI_CTRL.NULL;
      eInit                                       := E_PROGRESS.PROGRESS_BUSY;


    E_PROGRESS.PROGRESS_BUSY:
      GVL_NCI.stChannelCtrl[nChnInit].eCmd        := E_NCI_CTRL.INIT;

      IF (GVL_NCI.stChannelState[nChnInit].eState = E_NCI_STATE.INIT + E_PROGRESS.PROGRESS_ERROR)
      THEN
        eInit                                     := E_PROGRESS.PROGRESS_ERROR;

        stMsg.eType                               := E_MessageType.eMessageError;
        stMsg.eDevice                             := e_Device.NciChannelCtrl;
        stMsg.eSubdevice                          := e_SubDevice.NciStartUp;
        stMsg.iErrorNumber                        := nChnInit;

        stMsg.sText                               := concat('NCI.eInit ERROR at Index: ', TO_STRING(nChnInit));
        f_MessageSet(stMsg);

      ELSIF (GVL_NCI.stChannelState[nChnInit].eState = E_NCI_STATE.INIT + E_PROGRESS.PROGRESS_DONE)
      THEN
        eInit                                     := E_PROGRESS.PROGRESS_CHECK;
      END_IF


    E_PROGRESS.PROGRESS_CHECK:
      IF (nChnInit > PLC_CONSTANT.MAX_NCI_CH-1)
      THEN
        bInit                                     := TRUE;
        eInit                                     := E_PROGRESS.PROGRESS_DONE;

        stMsg.eType                               := E_MessageType.eMessageInfo;
        stMsg.eDevice                             := e_Device.NciChannelCtrl;
        stMsg.eSubdevice                          := e_SubDevice.NciStartUp;
        stMsg.iErrorNumber                        := MAX_NCI_CH;

        stMsg.sText                               := concat('NCI.eInit: ', TO_STRING(eInit));
        f_MessageSet(stMsg);

      ELSE
        nChnInit                                  := nChnInit + 1;
        eInit                                     := E_PROGRESS.PROGRESS_INIT;
      END_IF
  END_CASE
END_IF
//-----------------------------------------------------------------------------------------------------------------
// INIT/
//-----------------------------------------------------------------------------------------------------------------
//-----------------------------------------------------------------------------------------------------------------
//-----------------------------------------------------------------------------------------------------------------
// /CYCLE
//-----------------------------------------------------------------------------------------------------------------
FOR nChn := 1 TO MAX_NCI_CH
DO
  // call nci channel controller
  GVL_NCI.fbNciCtrl[nChn].Cycle();

  GVL_NCI.sProgNameActive[nChn]             := GVL_NCI.fbNciCtrl[nChn].ItfChannel.GetLoadedProg();
  GVL_NCI.fbNciCtrl[nChn].M_FunctionScope   := ADR(GVL_NCI.M_FunctionCyclic[nChn]);
END_FOR
//-----------------------------------------------------------------------------------------------------------------
// CYCLE/
//-----------------------------------------------------------------------------------------------------------------
//-----------------------------------------------------------------------------------------------------------------

END_PROGRAM

// ---- CAM.TcPOU
PROGRAM CAM
VAR
  bInit                     : BOOL;
  eInit                     : E_PROGRESS;

  nAxis,
  nAxisInit                 : UINT;

  stMsg                     : ST_Message;
END_VAR

//-----------------------------------------------------------------------------------------------------------------
// check if compiler define is present [PLC_STATE_DRIVE/CompilerDefines/Manual: CAM]
// see PLC_CONSTANT for conditional pragma
//-----------------------------------------------------------------------------------------------------------------
IF NOT PLC_CONSTANT.CAM_ACTIVE THEN eInit := E_PROGRESS.PROGRESS_NOT_EXIST; RETURN; END_IF
//-----------------------------------------------------------------------------------------------------------------
//-----------------------------------------------------------------------------------------------------------------
// check for MAIN.eInit
//-----------------------------------------------------------------------------------------------------------------
IF NOT (MAIN.eInit = E_PROGRESS.PROGRESS_DONE) THEN eInit   := E_PROGRESS.PROGRESS_INVALID; RETURN; END_IF
//-----------------------------------------------------------------------------------------------------------------
//-----------------------------------------------------------------------------------------------------------------
// /assign dataflow
//-----------------------------------------------------------------------------------------------------------------
FOR nAxis := 1 TO PLC_CONSTANT.MAX_AXIS
DO
  GVL_CAM.Control[nAxis].ItfMcAxes                := GVL_AXIS.ItfMcAxis;

  GVL_CAM.Control[nAxis].AxisIndex                := nAxis;

  GVL_CAM.Control[nAxis].AxisCtrl                 := ADR(GVL_CAM.Ctrl);          // command
  GVL_CAM.Control[nAxis].AxisState                := ADR(GVL_CAM.State);         // state + result of command

  GVL_CAM.Control[nAxis].Axes                     REF=   GVL_AXIS.AxisRef;        // All for one; coupling requires access across all axes

  GVL_CAM.Control[nAxis].AxisInfo                 := ADR(GVL_CAM.Info);
  GVL_CAM.Control[nAxis].AxisData                 := ADR(GVL_CAM.Data);

  GVL_CAM.Control[nAxis].MotionFunction           := ADR(GVL_CAM.MotionFunction);
  GVL_CAM.Control[nAxis].MotionFunctionPoint      := ADR(GVL_CAM.MotionFunctionPoint);
END_FOR
//-----------------------------------------------------------------------------------------------------------------
// assign dataflow/
//-----------------------------------------------------------------------------------------------------------------
//-----------------------------------------------------------------------------------------------------------------
// /INIT
//-----------------------------------------------------------------------------------------------------------------
IF NOT bInit
THEN
  CASE eInit
  OF
    E_PROGRESS.PROGRESS_INVALID,
    E_PROGRESS.PROGRESS_DONE:
      FOR nAxis := 1 TO PLC_CONSTANT.MAX_AXIS
      DO
        GVL_CAM.Control[nAxis].MessageLevel       := GVL_MSG.MessageLevelAxisCam;
      END_FOR
      nAxisInit                                   := 1;
      eInit                                       := E_PROGRESS.PROGRESS_INIT;


    E_PROGRESS.PROGRESS_INIT:
      stMsg.eType                                 := E_MessageType.eMessageVerbose;
      stMsg.eDevice                               := e_Device.Camming;
      stMsg.eSubdevice                            := e_SubDevice.CamStartUp;
      stMsg.iErrorNumber                          := nAxisInit;

      stMsg.sText                                 := concat('CAM.eInit: ', TO_STRING(eInit));

      IF (GVL_MSG.MessageLevelAxisCam = E_MessageType.eMessageVerbose)
      THEN
        f_MessageSet(stMsg);
      END_IF

      GVL_CAM.Ctrl[nAxisInit].eCmd               := E_AXIS_CTRL.AXIS_NULL;
      eInit                                       := E_PROGRESS.PROGRESS_BUSY;


    E_PROGRESS.PROGRESS_BUSY:
      GVL_CAM.Ctrl[nAxisInit].eCmd               := E_AXIS_CTRL.AXIS_INIT;

      IF (GVL_CAM.State[nAxisInit].eState = E_AXIS_STATE.AXIS_INIT + E_PROGRESS.PROGRESS_ERROR)
      THEN
        eInit                                     := E_PROGRESS.PROGRESS_ERROR;

        stMsg.eType                               := E_MessageType.eMessageError;
        stMsg.eDevice                             := e_Device.Camming;
        stMsg.eSubdevice                          := e_SubDevice.CamStartUp;
        stMsg.iErrorNumber                        := nAxisInit;

        stMsg.sText                               := concat('CAM.eInit ERROR at Index: ', TO_STRING(nAxisInit));
        f_MessageSet(stMsg);

      ELSIF (GVL_CAM.State[nAxisInit].eState = E_AXIS_STATE.AXIS_INIT + E_PROGRESS.PROGRESS_DONE)
      THEN
        eInit                                     := E_PROGRESS.PROGRESS_CHECK;
      END_IF


    E_PROGRESS.PROGRESS_CHECK:
      IF (nAxisInit > PLC_CONSTANT.MAX_AXIS-1)
      THEN
        bInit                                     := TRUE;
        eInit                                     := E_PROGRESS.PROGRESS_DONE;

        stMsg.eType                               := E_MessageType.eMessageInfo;
        stMsg.eDevice                             := e_Device.Camming;
        stMsg.eSubdevice                          := e_SubDevice.CamStartUp;
        stMsg.iErrorNumber                        := MAX_AXIS;

        stMsg.sText                               := concat('CAM.eInit: ', TO_STRING(eInit));
        f_MessageSet(stMsg);

      ELSE
        nAxisInit                                 := nAxisInit + 1;
        eInit                                     := E_PROGRESS.PROGRESS_INIT;
      END_IF
  END_CASE
END_IF
//-----------------------------------------------------------------------------------------------------------------
// INIT
//-----------------------------------------------------------------------------------------------------------------
//-----------------------------------------------------------------------------------------------------------------
// /cyclic
//-----------------------------------------------------------------------------------------------------------------
IF (eInit <> E_PROGRESS.PROGRESS_ERROR)
THEN
  FOR nAxis := 1 TO PLC_CONSTANT.MAX_AXIS
  DO
      GVL_CAM.Control[nAxis].Cycle();
  END_FOR
END_IF
//-----------------------------------------------------------------------------------------------------------------
// cyclic/
//-----------------------------------------------------------------------------------------------------------------

END_PROGRAM

// ---- MAPPING/MAPPING_out.TcPOU
PROGRAM MAPPING_out
VAR CONSTANT
{IF defined (AXIS_MAP)}
  {info 'MAPPING_out - AXIS_MAP'}
  bBypassMappingAxis        : BOOL  := FALSE;
{ELSE}
  bBypassMappingAxis        : BOOL  := TRUE;
{END_IF}
{IF defined (CAM_MAP)}
  {info 'MAPPING_out - CAM_MAP'}
  bBypassMappingCam         : BOOL  := FALSE;
{ELSE}
  bBypassMappingCam         : BOOL  := TRUE;
{END_IF}
{IF defined (TRIGGER_MAP)}
  {info 'MAPPING_out - TRIGGER_MAP'}
  bBypassMappingTrigger     : BOOL  := FALSE;
{ELSE}
  bBypassMappingTrigger     : BOOL  := TRUE;
{END_IF}
END_VAR
VAR
  bFirstCycle       : BOOL := TRUE;
{IF defined (AXIS_MAP)}
  AxisState         : U_AXIS_STATE;
  AxisInfo          : U_AXIS_INFO;
  AxisParameterRd   : U_AXIS_NC_PARAMETER_RD;
{ELSE}
  AxisState         : BYTE;
  AxisInfo          : BYTE;
  AxisParameterRd   : BYTE;
{END_IF}
{IF defined (CAM_MAP)}
  CamState          : U_CAM_STATE;
  CamData           : U_CAM_DATA;
  CamInfo           : U_CAM_INFO;
{ELSE}
  CamState          : BYTE;
  CamData           : BYTE;
  CamInfo           : BYTE;
{END_IF}
{IF defined (TRIGGER_MAP)}
  TriggerState      : U_TRIGGER_STATE;
  TouchProbeState   : U_TOUCH_PROBE_STATE;
{ELSE}
  TriggerState      : BYTE;
  TouchProbeState   : BYTE;
{END_IF}

  szAxisPara,
  szAxisInfo,
  szAxisState           : ARRAY[1..2] OF UDINT;

  szCamInfo,
  szCamData,
  szCamState            : ARRAY[1..2] OF UDINT;

  szStateTouchProbe,
  szStateTrigger	      :  ARRAY[1..2] OF UDINT;
END_VAR


IF (bFirstCycle)
THEN
  bFirstCycle         := FALSE;
  
  szAxisState[1]      := SIZEOF(AxisState);
  szAxisState[2]      := SIZEOF(GVL_AXIS.State);
  
  szAxisInfo [1]      := SIZEOF(AxisInfo);
  szAxisInfo [2]      := SIZEOF(GVL_AXIS.Info);
  
  szAxisPara [1]      := SIZEOF(AxisParameterRd);
  szAxisPara [2]      := SIZEOF(GVL_AXIS.NcParameterRd);
  
  
  szCamInfo  [1]      := SIZEOF(CamInfo);
  szCamInfo  [2]      := SIZEOF(GVL_CAM.Info);
  
  szCamData  [1]      := SIZEOF(CamData);
  szCamData  [2]      := SIZEOF(GVL_CAM.Data);
  
  szCamState [1]      := SIZEOF(CamState);
  szCamState [2]      := SIZEOF(GVL_CAM.State);
  
  szStateTrigger [1]  := SIZEOF(TriggerState);
  szStateTrigger [2]  := SIZEOF(GVL_FUNCTIONS.StateTrigger);
  
  szStateTouchProbe [1]  := SIZEOF(TouchProbeState);
  szStateTouchProbe [2]  := SIZEOF(GVL_FUNCTIONS.StateTouchProbe);
END_IF

IF NOT bBypassMappingAxis
THEN
  memcpy(ADR(AxisState),         ADR(GVL_AXIS.State),             SIZEOF(AxisState));
  memcpy(ADR(AxisInfo),          ADR(GVL_AXIS.Info),              SIZEOF(AxisInfo));
  memcpy(ADR(AxisParameterRd),   ADR(GVL_AXIS.NcParameterRd),     SIZEOF(AxisParameterRd));
END_IF

IF NOT bBypassMappingCam
THEN
  memcpy(ADR(CamInfo),    ADR(GVL_CAM.Info),    SIZEOF(CamInfo));
  memcpy(ADR(CamData),    ADR(GVL_CAM.Data),    SIZEOF(CamData));
  memcpy(ADR(CamState),   ADR(GVL_CAM.State),   SIZEOF(CamState));
END_IF

IF NOT bBypassMappingTrigger
THEN
  memcpy(ADR(TriggerState),     ADR(GVL_FUNCTIONS.StateTrigger),    SIZEOF(TriggerState));
  memcpy(ADR(TouchProbeState),  ADR(GVL_FUNCTIONS.StateTouchProbe), SIZEOF(TouchProbeState));
END_IF

END_PROGRAM

// ---- CAM/FB_CamCtrl.TcPOU
FUNCTION_BLOCK FB_CamCtrl EXTENDS FB_CamAxis IMPLEMENTS I_Cam_Ctrl
VAR
  _eInit                    : E_PROGRESS;
  _nAxisIndex               : UINT;       // know thyself

  // get interface from McAxis for access to Reset, Enable, Disable, Halt
  _ItfMcAxis                : ARRAY[1..PLC_CONSTANT.MAX_AXIS] OF I_McAxis;

  // pointers to all; access required for coupling; access by index
  _Axes                     : REFERENCE TO ARRAY[1..PLC_CONSTANT.MAX_AXIS] OF AXIS_REF;

  _Ctrl                     : POINTER TO ARRAY[1..PLC_CONSTANT.MAX_AXIS] OF ST_CAM_CTRL;    // contains command to be executed
  _State                    : POINTER TO ARRAY[1..PLC_CONSTANT.MAX_AXIS] OF ST_CAM_STATE;   // mirrors command with added result

  _Info                     : POINTER TO ARRAY[1..PLC_CONSTANT.MAX_AXIS] OF ST_CAM_INFO;    // Read Camming Info Data
  _Data                     : POINTER TO ARRAY[1..PLC_CONSTANT.MAX_AXIS] OF ST_CAM_DATA;    // Camming parameters

  _MotionFunction           : POINTER TO ARRAY[1..PLC_CONSTANT.MAX_AXIS] OF ST_MOTION_FUNCTION;
  _MotionFunctionPoint      : POINTER TO ARRAY[1..PLC_CONSTANT.MAX_AXIS] OF ST_MOTION_FUNCTION_POINT;

  // local copies of command
  _eCmd,
  _eCmdOld                       : E_AXIS_CTRL;

  // execution state
  _eResult                        : E_PROGRESS;   // result of execution state
  _eResultOld                     : E_PROGRESS;   // old result for detecting change
  _eState                         : E_AXIS_STATE; // execution state
END_VAR

PROPERTY Axes : reference TO ARRAY[1..PLC_CONSTANT.MAX_AXIS] OF AXIS_REF
SET
_Axes := Axes;
END_SET
END_PROPERTY

METHOD AxisCamIdle : E_PROGRESS
VAR_INPUT
  Execute           : BOOL;
END_VAR
VAR_INST
  _eResult,
  _eState           : E_PROGRESS;
  _stMsg            : ST_Message;
  _nRetry           : UINT;
END_VAR
IF NOT Execute THEN _eState := E_PROGRESS.PROGRESS_INIT; END_IF
IF NOT Check() THEN _eState := E_PROGRESS.PROGRESS_ERROR; END_IF

CASE _eState
OF
  E_PROGRESS.PROGRESS_INIT:
    IF Execute 
    THEN
      memset(ADR(_stMsg),0,SIZEOF(_stMsg));
      _nRetry                       := 0;
      _eResult                      := _ItfMcAxis[_nAxisIndex].Reset(FALSE);
      _eState                       := E_PROGRESS.PROGRESS_BUSY;
    END_IF
END_CASE
CASE _eState
OF
  E_PROGRESS.PROGRESS_PREPARE:
    _nRetry                         := _nRetry + 1;
    _eResult                        := _ItfMcAxis[_nAxisIndex].Reset(FALSE);
    _eResult                        := _ItfMcAxis[_nAxisIndex].Enable(FALSE);

    _eState                         := E_PROGRESS.PROGRESS_BUSY;

    _stMsg.eType                    := E_MessageType.eMessageInfo;
    _stMsg.eDevice                  := e_Device.Camming + (_AxisSlave.NcToPlc.AxisId);
    _stMsg.eSubdevice               :=  e_SubDevice.fbPower;
    _stMsg.iErrorNumber             := _nErrorId;

    _stMsg.sText                    := concat(TO_STRING(_eCmd), ' retry: ');
    _stMsg.sText                    := concat(_stMsg.sText, TO_STRING(_nRetry));

    IF (_MessageLevel < E_MessageType.eMessageError)
    THEN
      f_MessageSet(_stMsg);
    END_IF
END_CASE
CASE _eState
OF
  E_PROGRESS.PROGRESS_BUSY:
    _eResult                        := _ItfMcAxis[_nAxisIndex].Reset(TRUE);

    IF (_eResult = E_PROGRESS.PROGRESS_DONE)
    THEN
      _eState                       := E_PROGRESS.PROGRESS_STARTUP;
    END_IF
END_CASE
CASE _eState
OF
  E_PROGRESS.PROGRESS_STARTUP:
    _eResult                        := _ItfMcAxis[_nAxisIndex].Reset(FALSE);
    _eResult                        := _ItfMcAxis[_nAxisIndex].Enable(FALSE);
    _eState                         := E_PROGRESS.PROGRESS_CHECK;
END_CASE
CASE _eState
OF
  E_PROGRESS.PROGRESS_CHECK:
    _eResult                        := _ItfMcAxis[_nAxisIndex].Enable(TRUE);

    IF (_nRetry > MAX_RETRY)
    THEN
      _eState                       := E_PROGRESS.PROGRESS_ERROR;

    ELSIF (_eResult = E_PROGRESS.PROGRESS_DONE)
    THEN
      _ItfMcAxis[_nAxisIndex].Enable(FALSE);
      _eState                       := E_PROGRESS.PROGRESS_DONE;

    ELSIF (_eResult = E_PROGRESS.PROGRESS_ERROR)
    THEN
      _eState                       := E_PROGRESS.PROGRESS_PREPARE;

      _nErrorId                     := _AxisSlave.NcToPlc.ErrorCode;
    
      _stMsg.eType                  := E_MessageType.eMessageError;
      _stMsg.eDevice                := e_Device.Camming + (_AxisSlave.NcToPlc.AxisId);
      _stMsg.eSubdevice             :=  e_SubDevice.fbPower;
      _stMsg.iErrorNumber           := _nErrorId;

      _stMsg.sText                  := concat(TO_STRING(_eCmd), ' error axis enable: ');
      _stMsg.sText                  := concat(_stMsg.sText, TO_STRING(_nAxisIndex));

      f_MessageSet(_stMsg);
    END_IF
END_CASE

AxisCamIdle                                := _eState;
END_METHOD

METHOD AxisCamIn : E_PROGRESS
VAR_INPUT
  Execute           : BOOL;
END_VAR
VAR_INST
  _eCk              : E_CHECK_STATE;

  _eResult,
  _eState           : E_PROGRESS;
  _rValue           : LREAL;
  _udiErr           : UDINT;
  _stMsg            : ST_Message;

END_VAR
IF NOT Execute THEN _eState := E_PROGRESS.PROGRESS_INIT; END_IF
IF NOT Check() THEN _eState := E_PROGRESS.PROGRESS_ERROR; END_IF


CASE _eState
OF
  E_PROGRESS.PROGRESS_INIT:
    IF Execute 
    THEN
      memset(ADR(_stMsg),0,SIZEOF(_stMsg));
      _udiErr                       := 0;

      IF NOT (_stCamData.nMasterIndex > 0) OR
         NOT (_stCamData.nMasterIndex < PLC_CONSTANT.MAX_AXIS+1)
      THEN
        _eState                     := E_PROGRESS.PROGRESS_ERROR;
        _eCk                        := E_CHECK_STATE.CAM_MASTER_AXIS_REF_INVALID;

        _stMsg.eType                := E_MessageType.eMessageError;
        _stMsg.eDevice              := E_Device.Camming + (_AxisSlave.NcToPlc.AxisId);
        _stMsg.eSubdevice           := e_Subdevice.CamControl;
        _stMsg.iErrorNumber         := _stCamData.nMasterIndex;
  
        _stMsg.sText                := concat(' : ', TO_STRING(_eCk));
        f_MessageSet(_stMsg);

      ELSE
        _eState                     := E_PROGRESS.PROGRESS_BUSY;
        _eCk                        := E_CHECK_STATE.CHECK_DONE;
        _eResult                    := CamIn(FALSE, _stCamData.nMasterIndex);
      END_IF
    END_IF
END_CASE
CASE _eState
OF
  E_PROGRESS.PROGRESS_BUSY:
      _eResult                      := CamIn(TRUE, _stCamData.nMasterIndex);

    IF (_eResult = E_PROGRESS.PROGRESS_ERROR)
    THEN
      CamIn(FALSE, _stCamData.nMasterIndex);
      _eState                       := E_PROGRESS.PROGRESS_ERROR;
      _udiErr                       := _fbCamInV2.ErrorID;

    ELSIF (_eResult = E_PROGRESS.PROGRESS_DONE)
    THEN
      CamIn(FALSE, _stCamData.nMasterIndex);
      _eState                       := E_PROGRESS.PROGRESS_DONE;
    END_IF
END_CASE


AxisCamIn                           := _eState;
END_METHOD

METHOD AxisCamInfo : E_PROGRESS
VAR_INPUT
  Execute           : BOOL;
END_VAR
VAR_INST
  _eCk              : E_CHECK_STATE;

  _eResult,
  _eState           : E_PROGRESS;
  _rValue           : LREAL;
  _udiErr           : UDINT;
  _stMsg            : ST_Message;

END_VAR
IF NOT Execute THEN _eState := E_PROGRESS.PROGRESS_INIT; END_IF
IF NOT Check() THEN _eState := E_PROGRESS.PROGRESS_ERROR; END_IF


CASE _eState
OF
  E_PROGRESS.PROGRESS_INIT:
    IF Execute 
    THEN
      memset(ADR(_stMsg),0,SIZEOF(_stMsg));
      _udiErr                       := 0;

      _eState                       := E_PROGRESS.PROGRESS_BUSY;
      _eCk                          := E_CHECK_STATE.CHECK_DONE;
      _eResult                      := CamInfo(FALSE, _stCamData.nCamTableId, _stCamData.bAtMasterPosition, _stCamData.rMasterPosition);
    END_IF
END_CASE
CASE _eState
OF
  E_PROGRESS.PROGRESS_BUSY:
      _eResult                      := CamInfo(TRUE, _stCamData.nCamTableId, _stCamData.bAtMasterPosition, _stCamData.rMasterPosition);

    IF (_eResult = E_PROGRESS.PROGRESS_ERROR)
    THEN
      _eState                       := E_PROGRESS.PROGRESS_ERROR;
      CamInfo(FALSE, _stCamData.nCamTableId, _stCamData.bAtMasterPosition, _stCamData.rMasterPosition);

    ELSIF (_eResult = E_PROGRESS.PROGRESS_DONE)
    THEN
      _eState                       := E_PROGRESS.PROGRESS_CHECK;
      CamInfo(FALSE, _stCamData.nCamTableId, _stCamData.bAtMasterPosition, _stCamData.rMasterPosition);
    END_IF
END_CASE
CASE _eState
OF
  E_PROGRESS.PROGRESS_CHECK:
    _Info^[_nAxisIndex]             := CamInfoData;

    _stMsg.eType                    := E_MessageType.eMessageInfo;
    _stMsg.eDevice                  := E_Device.Camming + (_AxisSlave.NcToPlc.AxisId);
    _stMsg.eSubdevice               := e_Subdevice.CamControl;
    _stMsg.iErrorNumber             := 0;

    _stMsg.sText                    := concat('CamInfoData : ', TO_STRING(_eState));

    IF (_MessageLevel < E_MessageType.eMessageError)
    THEN
      f_MessageSet(_stMsg);
    END_IF

    _eState                         := E_PROGRESS.PROGRESS_DONE;
END_CASE


AxisCamInfo                         := _eState;
END_METHOD

METHOD AxisCamOut : E_PROGRESS
VAR_INPUT
  Execute           : BOOL;
END_VAR
VAR_INST
  _eResult,
  _eState           : E_PROGRESS;
END_VAR
IF NOT Execute THEN _eState := E_PROGRESS.PROGRESS_INIT; END_IF
IF NOT Check() THEN _eState := E_PROGRESS.PROGRESS_ERROR; END_IF


CASE _eState
OF
  E_PROGRESS.PROGRESS_INIT:
    IF Execute 
    THEN
      _eState                       := E_PROGRESS.PROGRESS_BUSY;
      _eResult                      := CamOut(FALSE);
    END_IF
END_CASE
CASE _eState
OF
  E_PROGRESS.PROGRESS_BUSY:
    _eResult                        := CamOut(TRUE);

    IF (_eResult = E_PROGRESS.PROGRESS_ERROR)
    THEN
      CamOut(FALSE);
      _eState                       := E_PROGRESS.PROGRESS_ERROR;

    ELSIF (_eResult = E_PROGRESS.PROGRESS_DONE)
    THEN
      CamOut(FALSE);
      _eState                       := E_PROGRESS.PROGRESS_DONE;
    END_IF
END_CASE


AxisCamOut                          := _eState;
END_METHOD

METHOD AxisCamScaling : E_PROGRESS
VAR_INPUT
  Execute             : BOOL;
END_VAR
VAR_INST
  _eResult,
  _eState             : E_PROGRESS;
  _rValue             : LREAL;
  _udiErr             : UDINT;
  _stMsg              : ST_Message;
END_VAR

IF NOT __ISVALIDREF(_AxisSlave)
THEN
  _eCheck                   := E_CHECK_STATE.CAM_SLAVE_AXIS_REF_INVALID;
  AxisCamScaling            := E_PROGRESS.PROGRESS_ERROR;
  RETURN;
END_IF

IF NOT Execute THEN _eState := E_PROGRESS.PROGRESS_INIT; END_IF

CASE _eState
OF
  E_PROGRESS.PROGRESS_INIT:
    IF Execute 
    THEN
      memset(ADR(_stMsg),0,SIZEOF(_stMsg));
      _udiErr               := 0;
      _rValue               := 0;
      _eState               := E_PROGRESS.PROGRESS_BUSY;
      _eResult              := CamScaling(FALSE);
    END_IF
END_CASE
CASE _eState
OF
  E_PROGRESS.PROGRESS_BUSY:
    _eResult                := CamScaling(TRUE);
    IF (_eResult = E_PROGRESS.PROGRESS_ERROR)
    THEN
      CamScaling(FALSE);
      _eState               := E_PROGRESS.PROGRESS_ERROR;

    ELSIF (_eResult = E_PROGRESS.PROGRESS_DONE)
    THEN
      CamScaling(FALSE);
      _eState               := E_PROGRESS.PROGRESS_DONE;
    END_IF
END_CASE

AxisCamScaling              := _eState;
END_METHOD

PROPERTY AxisCtrl : pointer to ARRAY[1..PLC_CONSTANT.MAX_AXIS] OF st_axis_ctrl
SET
_Ctrl := AxisCtrl;
END_SET
END_PROPERTY

PROPERTY AxisData : pointer to ARRAY[1..PLC_CONSTANT.MAX_AXIS] OF ST_CAM_DATA
SET
_Data := AxisData;
END_SET
END_PROPERTY

PROPERTY AxisIndex : uint
SET
_nAxisIndex := AxisIndex;
END_SET
END_PROPERTY

PROPERTY AxisInfo : pointer to ARRAY[1..PLC_CONSTANT.MAX_AXIS] OF ST_AXIS_INFO
SET
_Info := AxisInfo;
END_SET
END_PROPERTY

METHOD AxisReadMotionFunction : E_PROGRESS
VAR_INPUT
  Execute             : BOOL;
END_VAR
VAR_INST
  _eResult,
  _eState             : E_PROGRESS;
  _rValue             : LREAL;
  _udiErr             : UDINT;
  _stMsg              : ST_Message;
END_VAR

IF NOT __ISVALIDREF(_AxisSlave)
THEN
  _eCheck                   := E_CHECK_STATE.CAM_SLAVE_AXIS_REF_INVALID;
  AxisReadMotionFunction    := E_PROGRESS.PROGRESS_ERROR;
  RETURN;
END_IF

IF NOT Execute THEN _eState := E_PROGRESS.PROGRESS_INIT; END_IF

CASE _eState
OF
  E_PROGRESS.PROGRESS_INIT:
    IF Execute 
    THEN
      memset(ADR(_stMsg),0,SIZEOF(_stMsg));
      _udiErr               := 0;
      _rValue               := 0;
      _eState               := E_PROGRESS.PROGRESS_BUSY;
      _eResult              := ReadMotionFunction(FALSE);
    END_IF
END_CASE
CASE _eState
OF
  E_PROGRESS.PROGRESS_BUSY:
    _eResult                := ReadMotionFunction(TRUE);
    IF (_eResult = E_PROGRESS.PROGRESS_ERROR)
    THEN
      ReadMotionFunction(FALSE);
      _eState               := E_PROGRESS.PROGRESS_ERROR;

    ELSIF (_eResult = E_PROGRESS.PROGRESS_DONE)
    THEN
      ReadMotionFunction(FALSE);
      _MotionFunction^[_nAxisIndex]     := ReadMotionFunctionData;
      _eState                           := E_PROGRESS.PROGRESS_DONE;
    END_IF
END_CASE

AxisReadMotionFunction      := _eState;
END_METHOD

METHOD AxisReadMotionFunctionPoint : E_PROGRESS
VAR_INPUT
  Execute             : BOOL;
END_VAR
VAR_INST
  _eResult,
  _eState             : E_PROGRESS;
  _rValue             : LREAL;
  _udiErr             : UDINT;
  _stMsg              : ST_Message;
END_VAR

IF NOT __ISVALIDREF(_AxisSlave)
THEN
  _eCheck                       := E_CHECK_STATE.CAM_SLAVE_AXIS_REF_INVALID;
  AxisReadMotionFunctionPoint   := E_PROGRESS.PROGRESS_ERROR;
  RETURN;
END_IF

IF NOT Execute THEN _eState := E_PROGRESS.PROGRESS_INIT; END_IF

CASE _eState
OF
  E_PROGRESS.PROGRESS_INIT:
    IF Execute 
    THEN
      memset(ADR(_stMsg),0,SIZEOF(_stMsg));
      _udiErr               := 0;
      _rValue               := 0;
      _eState               := E_PROGRESS.PROGRESS_BUSY;
      _eResult              := ReadMotionFunctionPoint(FALSE);
    END_IF
END_CASE
CASE _eState
OF
  E_PROGRESS.PROGRESS_BUSY:
    _eResult                := ReadMotionFunctionPoint(TRUE);
    IF (_eResult = E_PROGRESS.PROGRESS_ERROR)
    THEN
      ReadMotionFunctionPoint(FALSE);
      _eState               := E_PROGRESS.PROGRESS_ERROR;

    ELSIF (_eResult = E_PROGRESS.PROGRESS_DONE)
    THEN
      ReadMotionFunctionPoint(FALSE);
      _MotionFunctionPoint^[_nAxisIndex]  := ReadMotionFunctionPointData;
      _eState                             := E_PROGRESS.PROGRESS_DONE;
    END_IF
END_CASE

AxisReadMotionFunctionPoint      := _eState;
END_METHOD

PROPERTY AxisState : pointer to ARRAY[1..PLC_CONSTANT.MAX_AXIS] OF ST_CAM_STATE
SET
_State := AxisState;
END_SET
END_PROPERTY

METHOD AxisWriteMotionFunction : E_PROGRESS
VAR_INPUT
  Execute             : BOOL;
END_VAR
VAR_INST
  _eResult,
  _eState             : E_PROGRESS;
  _rValue             : LREAL;
  _udiErr             : UDINT;
  _stMsg              : ST_Message;
END_VAR

IF NOT __ISVALIDREF(_AxisSlave)
THEN
  _eCheck                       := E_CHECK_STATE.CAM_SLAVE_AXIS_REF_INVALID;
  AxisWriteMotionFunction       := E_PROGRESS.PROGRESS_ERROR;
  RETURN;
END_IF

IF NOT Execute THEN _eState := E_PROGRESS.PROGRESS_INIT; END_IF

CASE _eState
OF
  E_PROGRESS.PROGRESS_INIT:
    IF Execute 
    THEN
      memset(ADR(_stMsg),0,SIZEOF(_stMsg));
      _udiErr               := 0;
      _rValue               := 0;
      _eState               := E_PROGRESS.PROGRESS_BUSY;
      _eResult              := WriteMotionFunction(FALSE);
    END_IF
END_CASE
CASE _eState
OF
  E_PROGRESS.PROGRESS_BUSY:
    _eResult                := WriteMotionFunction(TRUE);
    IF (_eResult = E_PROGRESS.PROGRESS_ERROR)
    THEN
      WriteMotionFunction(FALSE);
      _eState               := E_PROGRESS.PROGRESS_ERROR;

    ELSIF (_eResult = E_PROGRESS.PROGRESS_DONE)
    THEN
      WriteMotionFunction(FALSE);
      _eState                             := E_PROGRESS.PROGRESS_DONE;
    END_IF
END_CASE

AxisWriteMotionFunction     := _eState;
END_METHOD

METHOD AxisWriteMotionFunctionPoint : E_PROGRESS
VAR_INPUT
  Execute             : BOOL;
END_VAR
VAR_INST
  _eResult,
  _eState             : E_PROGRESS;
  _rValue             : LREAL;
  _udiErr             : UDINT;
  _stMsg              : ST_Message;
END_VAR

IF NOT __ISVALIDREF(_AxisSlave)
THEN
  _eCheck                       := E_CHECK_STATE.CAM_SLAVE_AXIS_REF_INVALID;
  AxisWriteMotionFunctionPoint  := E_PROGRESS.PROGRESS_ERROR;
  RETURN;
END_IF

IF NOT Execute THEN _eState := E_PROGRESS.PROGRESS_INIT; END_IF

CASE _eState
OF
  E_PROGRESS.PROGRESS_INIT:
    IF Execute 
    THEN
      memset(ADR(_stMsg),0,SIZEOF(_stMsg));
      _udiErr               := 0;
      _rValue               := 0;
      _eState               := E_PROGRESS.PROGRESS_BUSY;
      _eResult              := WriteMotionFunctionPoint(FALSE);
    END_IF
END_CASE
CASE _eState
OF
  E_PROGRESS.PROGRESS_BUSY:
    _eResult                := WriteMotionFunctionPoint(TRUE);
    IF (_eResult = E_PROGRESS.PROGRESS_ERROR)
    THEN
      WriteMotionFunctionPoint(FALSE);
      _eState               := E_PROGRESS.PROGRESS_ERROR;

    ELSIF (_eResult = E_PROGRESS.PROGRESS_DONE)
    THEN
      WriteMotionFunctionPoint(FALSE);
      _eState               := E_PROGRESS.PROGRESS_DONE;
    END_IF
END_CASE

AxisWriteMotionFunctionPoint := _eState;
END_METHOD

METHOD PRIVATE CamInit : E_PROGRESS
VAR_INPUT
  Execute           : BOOL;
END_VAR
VAR_INST
  _eResult,
  _eState           : E_PROGRESS;
  _rValue           : LREAL;
  _stMsg            : ST_Message;
END_VAR
IF NOT Check() THEN _eState := E_PROGRESS.PROGRESS_ERROR; END_IF
IF NOT Execute THEN _eState := E_PROGRESS.PROGRESS_INIT; END_IF

CASE _eState
OF
  E_PROGRESS.PROGRESS_INIT:
    IF Execute 
    THEN
      memset(ADR(_stMsg),0,SIZEOF(_stMsg));

      _nErrorId                     := 0;
      _rValue                       := 0;
      _eState                       := E_PROGRESS.PROGRESS_BUSY;
      _eInit                        := _eState;
    END_IF
END_CASE
CASE _eState
OF
  E_PROGRESS.PROGRESS_BUSY:
    _eState                         := E_PROGRESS.PROGRESS_STARTUP;
END_CASE
CASE _eState
OF
  E_PROGRESS.PROGRESS_STARTUP:
    // keep this for future use
    _eResult                        := E_PROGRESS.PROGRESS_DONE;//StartUp(TRUE);
    IF (_eResult = E_PROGRESS.PROGRESS_DONE)
    THEN
      _eState                       := E_PROGRESS.PROGRESS_PREPARE;
      _ItfMcAxis[_nAxisIndex].Reset(FALSE);
    ELSIF (_eResult = E_PROGRESS.PROGRESS_ERROR)
    THEN
      _eState                       := _eResult;

      _stMsg.eType                  := E_MessageType.eMessageError;
      _stMsg.eDevice                := e_Device.Camming + (_AxisSlave.NcToPlc.AxisId);
      _stMsg.eSubdevice             := e_Subdevice.CamStartUp;
      _stMsg.iErrorNumber := _nErrorId  := 6666;

      _stMsg.sText                  := TO_STRING(_eState);
      f_MessageSet(_stMsg);
    END_IF
END_CASE
CASE _eState
OF
  E_PROGRESS.PROGRESS_PREPARE:
    _eResult                        := _ItfMcAxis[_nAxisIndex].Reset(TRUE);
    IF (_eResult = E_PROGRESS.PROGRESS_DONE)
    THEN
      _eState                       := E_PROGRESS.PROGRESS_WORKING;
    ELSIF (_eResult = E_PROGRESS.PROGRESS_ERROR)
    THEN
      _eState                       := _eResult;

      _stMsg.eType                  := E_MessageType.eMessageError;
      _stMsg.eDevice                := e_Device.Camming + (_AxisSlave.NcToPlc.AxisId);
      _stMsg.eSubdevice             := e_Subdevice.fbReset;
      _stMsg.iErrorNumber           := _AxisSlave.Status.ErrorID;

      _stMsg.sText                  := TO_STRING(_eState);
      f_MessageSet(_stMsg);
    END_IF
END_CASE
CASE _eState
OF
  E_PROGRESS.PROGRESS_CHECK:
    _eResult                        := _ItfMcAxis[_nAxisIndex].Reset(FALSE);
    _eState                         := E_PROGRESS.PROGRESS_OCCUPIED;
END_CASE
CASE _eState
OF
  E_PROGRESS.PROGRESS_OCCUPIED:
    _eState                         := E_PROGRESS.PROGRESS_WORKING;
END_CASE
CASE _eState
OF
  E_PROGRESS.PROGRESS_WORKING:
    _eState                         := E_PROGRESS.PROGRESS_DONE;

    _stMsg.eType                    := E_MessageType.eMessageInfo;
    _stMsg.eDevice                  := e_Device.Camming + (_AxisSlave.NcToPlc.AxisId);
    _stMsg.eSubdevice               := e_Subdevice.CamControl;
    _stMsg.iErrorNumber             := 0;
    _stMsg.sText                    := concat('CamInit: ', TO_STRING(_eState));

    IF (_MessageLevel < E_MessageType.eMessageError)
    THEN
      f_MessageSet(_stMsg);
    END_IF
END_CASE

CamInit                            := _eState;
END_METHOD

METHOD PRIVATE Check : BOOL

//-----------------------------------------------------------------------------
IF (_nAxisIndex < 1) OR
   (_nAxisIndex > PLC_CONSTANT.MAX_AXIS)
THEN
  _eCheck                 := E_CHECK_STATE.AXIS_INDEX_OUT_OF_RANGE;
  RETURN;
END_IF
//-----------------------------------------------------------------------------
// get my AXIS_REF pointer for use in base class
//-----------------------------------------------------------------------------
_AxisSlave                := _Axes[_nAxisIndex];
//-----------------------------------------------------------------------------

IF NOT (_ItfMcAxis[_nAxisIndex] <> 0)
THEN
  _eCheck                 := E_CHECK_STATE.CAM_SLAVE_ITF_MC_AXIS_INVALID;
  RETURN;
END_IF


IF NOT (_Ctrl <> 0)
THEN
  _eCheck                 := E_CHECK_STATE.AXIS_CTRL_POINTER_INVALID;
  RETURN;
END_IF

IF NOT (_State <> 0)
THEN
  _eCheck                 := E_CHECK_STATE.AXIS_STATE_POINTER_INVALID;
  RETURN;
END_IF

IF NOT (_Info <> 0)
THEN
  _eCheck                 := E_CHECK_STATE.AXIS_INFO_POINTER_INVALID;
  RETURN;
END_IF

IF NOT (_Data <> 0)
THEN
  _eCheck                 := E_CHECK_STATE.AXIS_DATA_POINTER_INVALID;
  RETURN;
END_IF

IF NOT (_MotionFunction <> 0)
THEN
  _eCheck                 := E_CHECK_STATE.CAM_MOTION_FUNCTION_POINTER_INVALID;
  RETURN;
END_IF

IF NOT (_MotionFunctionPoint <> 0)
THEN
  _eCheck                 := E_CHECK_STATE.CAM_MOTION_FUNCTION_POINT_POINTER_INVALID;
  RETURN;
END_IF


//-----------------------------------------------------------------------------
//  NaN INF check
//-----------------------------------------------------------------------------
IF NOT IsFinite(F_LReal(_Data^[_nAxisIndex].rActivationPosition))
THEN
  _Data^[_nAxisIndex].rActivationPosition               := 0.0;
END_IF

IF NOT IsFinite(F_LReal(_Data^[_nAxisIndex].stCamScalingData.rMasterOffset))
THEN
  _Data^[_nAxisIndex].stCamScalingData.rMasterOffset    := 0.0;
END_IF

IF NOT IsFinite(F_LReal(_Data^[_nAxisIndex].stCamScalingData.rMasterScaling))
THEN
  _Data^[_nAxisIndex].stCamScalingData.rMasterScaling   := 0.0;
END_IF

IF NOT IsFinite(F_LReal(_Data^[_nAxisIndex].stCamScalingData.rSlaveOffset))
THEN
  _Data^[_nAxisIndex].stCamScalingData.rSlaveOffset     := 0.0;
END_IF

IF NOT IsFinite(F_LReal(_Data^[_nAxisIndex].stCamScalingData.rSlaveScaling))
THEN
	_Data^[_nAxisIndex].stCamScalingData.rSlaveScaling   := 0.0;
END_IF
//-----------------------------------------------------------------------------
//-----------------------------------------------------------------------------
_eCheck                   := E_CHECK_STATE.CHECK_DONE;
Check                     := TRUE;
//-----------------------------------------------------------------------------
//-----------------------------------------------------------------------------
END_METHOD

//-------------------------------------------------------------------------------------
//
//  HAUD 2024 01 20
//
//  Cmd
//    - gets state for ctrl
//    - checks for eInit to be done, before any other commands are accepted
//    - prepare your commands here
//    - init what you have to here
//
//-------------------------------------------------------------------------------------
METHOD PRIVATE Cmd  : E_AXIS_STATE
VAR_INPUT
  eCmd              : E_AXIS_CTRL;
END_VAR
VAR_INST
  _IdxMaster        : UINT;
  _stMsg            : ST_Message;
  _estate           : E_AXIS_STATE;
END_VAR
CASE eCmd
OF
  //-------------------------------------------------------------------------------------
  E_AXIS_CTRL.CAM_INIT:
    _eInit    := _eResult             := CamInit(FALSE);
    _estate                           := E_AXIS_STATE.CAM_INIT;
ELSE
  IF (_eInit <> E_PROGRESS.PROGRESS_DONE)
  THEN
    _eResult                          := E_PROGRESS.PROGRESS_INVALID;
    _estate                           := E_AXIS_STATE.AXIS_NO_INIT;
  ELSE
    CASE eCmd
    OF
      //---------------------------------------------------------------------------------
      E_AXIS_CTRL.AXIS_IDLE:
        _eResult                      := AxisCamIdle(FALSE);
        _estate                       := E_AXIS_STATE.AXIS_IDLE;

      //---------------------------------------------------------------------------------
      E_AXIS_CTRL.CAM_IN:
        _IdxMaster                    := _Data^[_nAxisIndex].nMasterIndex;
        _stCamData                    := _Data^[_nAxisIndex];
        _eResult                      := AxisCamIn(FALSE);
        _estate                       := E_AXIS_STATE.CAM_IN;

      //---------------------------------------------------------------------------------
      E_AXIS_CTRL.CAM_OUT:
        _eResult                      := AxisCamOut(FALSE);
        _estate                       := E_AXIS_STATE.CAM_OUT;

      //---------------------------------------------------------------------------------
      E_AXIS_CTRL.CAM_SCALING:
        _stCamData                    := _Data^[_nAxisIndex];
        _eResult                      := AxisCamScaling(FALSE);
        _eState                       := E_AXIS_STATE.CAM_SCALING;

      //---------------------------------------------------------------------------------
      E_AXIS_CTRL.CAM_INFO:
        _eResult                      := AxisCamInfo(FALSE);
        _estate                       := E_AXIS_STATE.CAM_INFO;

      //---------------------------------------------------------------------------------
      E_AXIS_CTRL.CAM_RD_MOTION_FUNCTION:
        _eResult                      := AxisReadMotionFunction(FALSE);
        _stCamData                    := _Data^[_nAxisIndex];
        _estate                       := E_AXIS_STATE.CAM_RD_MOTION_FUNCTION;

      //---------------------------------------------------------------------------------
      E_AXIS_CTRL.CAM_RD_MOTION_FUNCTION_POINT:
        _eResult                      := AxisReadMotionFunctionPoint(FALSE);
        _stCamData                    := _Data^[_nAxisIndex];
        _estate                       := E_AXIS_STATE.CAM_RD_MOTION_FUNCTION_POINT;

      //---------------------------------------------------------------------------------
      E_AXIS_CTRL.CAM_RD_MOTION_FUNCTIONS_VALUES:
        _stCamData                    := _Data^[_nAxisIndex];
        _estate                       := E_AXIS_STATE.CAM_RD_MOTION_FUNCTIONS_VALUES;

      //---------------------------------------------------------------------------------
      E_AXIS_CTRL.CAM_WRT_MOTION_FUNCTION:
        _eResult                      := AxisWriteMotionFunction(FALSE);
        _stCamData                    := _Data^[_nAxisIndex];
        WriteMotionFunctionData       := _MotionFunction^[_nAxisIndex];
        _estate                       := E_AXIS_STATE.CAM_WRT_MOTION_FUNCTION;

      //---------------------------------------------------------------------------------
      E_AXIS_CTRL.CAM_WRT_MOTION_FUNCTION_POINT:
        _eResult                      := AxisWriteMotionFunctionPoint(FALSE);
        _stCamData                    := _Data^[_nAxisIndex];
        WriteMotionFunctionPointData  := _MotionFunctionPoint^[_nAxisIndex];
        _estate                       := E_AXIS_STATE.CAM_WRT_MOTION_FUNCTION_POINT;

    //-----------------------------------------------------------------------------------
    ELSE
      _estate                         := E_AXIS_STATE.AXIS_NULL;

      IF (eCmd = E_AXIS_CTRL.AXIS_NULL)
      THEN
        _eResult                      := E_PROGRESS.PROGRESS_DONE;
      ELSE
        _eResult                      := E_PROGRESS.PROGRESS_INVALID;
  
        _stMsg.eType                  := E_MessageType.eMessageError;
        _stMsg.eDevice                := E_Device.Camming + (_AxisSlave.NcToPlc.AxisId);
        _stMsg.eSubdevice             := e_Subdevice.CamControl;
        _stMsg.iErrorNumber           := 0;
  
        _stMsg.sText                  := 'E_AXIS_CTRL.';
        _stMsg.sText                  := concat(_stMsg.sText, TO_STRING(eCmd));
        _stMsg.sText                  := concat(_stMsg.sText, ': ');
        _stMsg.sText                  := concat(_stMsg.sText, TO_STRING(_eResult));

        f_MessageSet(_stMsg);
      END_IF
    END_CASE
  END_IF // _eInit
END_CASE

Cmd                                   := _estate;
END_METHOD

PROPERTY CouplingState : array[0..7] of word
GET
VAR
  wtmp      : ARRAY[0..7] OF WORD;
END_VAR

memcpy(ADR(wtmp[0]) , ADR(_AxisSlave.NcToPlc.CamCouplingState[0]), 1);
memcpy(ADR(wtmp[1]) , ADR(_AxisSlave.NcToPlc.CamCouplingState[1]), 1);
memcpy(ADR(wtmp[2]) , ADR(_AxisSlave.NcToPlc.CamCouplingState[2]), 1);
memcpy(ADR(wtmp[3]) , ADR(_AxisSlave.NcToPlc.CamCouplingState[3]), 1);
memcpy(ADR(wtmp[4]) , ADR(_AxisSlave.NcToPlc.CamCouplingState[4]), 1);
memcpy(ADR(wtmp[5]) , ADR(_AxisSlave.NcToPlc.CamCouplingState[5]), 1);
memcpy(ADR(wtmp[6]) , ADR(_AxisSlave.NcToPlc.CamCouplingState[6]), 1);
memcpy(ADR(wtmp[7]) , ADR(_AxisSlave.NcToPlc.CamCouplingState[7]), 1);

CouplingState := wtmp;
END_GET
END_PROPERTY

METHOD Cycle  : e_progress
VAR_INST
  _eCycle     : E_PROGRESS;

  _eCheckOld  : E_CHECK_STATE;
END_VAR
IF NOT Check() THEN Cycle := _eCycle := _eResult := E_PROGRESS.PROGRESS_ERROR; END_IF
//-----------------------------------------------------------------------------
//-----------------------------------------------------------------------------
// OnChange log _eCheck; in case of error --> return to caller
//-----------------------------------------------------------------------------
IF (_eCheck <> _eCheckOld)
THEN
  LogCheck();
  _eCheckOld                        := _eCheck;
END_IF
//-----------------------------------------------------------------------------
IF NOT (_eCheck = E_CHECK_STATE.CHECK_DONE)
THEN
  RETURN;
END_IF
//-----------------------------------------------------------------------------
//-----------------------------------------------------------------------------
// get command from outside world
//-----------------------------------------------------------------------------
_eCmd                              := _Ctrl^[_nAxisIndex].eCmd;
//-----------------------------------------------------------------------------
//-----------------------------------------------------------------------------
//  OnChange react to command
//-----------------------------------------------------------------------------
IF (_eCmd <> _eCmdOld)
THEN
  // get busy
  _eState                           := Cmd(_eCmd); // get execution state for command
  _eCmdOld                         := _eCmd;
  LogControl();
END_IF
//-----------------------------------------------------------------------------
//-----------------------------------------------------------------------------
//  execution result
//-----------------------------------------------------------------------------
CASE _eResult
OF
  E_PROGRESS.PROGRESS_INVALID:
    _State^[_nAxisIndex].eState     := TO_UINT(E_PROGRESS.PROGRESS_ERROR);

  E_PROGRESS.PROGRESS_ERROR:
    _State^[_nAxisIndex].eState     := _eState + E_PROGRESS.PROGRESS_ERROR;

  E_PROGRESS.PROGRESS_DONE:
    _State^[_nAxisIndex].eState     := _eState + E_PROGRESS.PROGRESS_DONE;

ELSE
    _State^[_nAxisIndex].eState     := _eState + _eResult;
  //-----------------------------------------------------------------------------
  //-----------------------------------------------------------------------------
  //  execution state for command
  //-----------------------------------------------------------------------------
  CASE _eState
  OF
    //---------------------------------------------------------------------------
    E_AXIS_STATE.AXIS_INIT:
      // axis always requires one init from outside world at startup
      // _eInit has to be valid for other commands to be accepted in Cmd(_eCtrl)
      _eInit := _eResult            := CamInit(TRUE);
  
    //---------------------------------------------------------------------------
    E_AXIS_STATE.AXIS_NO_INIT:
      // we are here because you sent a command before having done CAM_INIT
      _eResult                      := E_PROGRESS.PROGRESS_ERROR;
  
    //---------------------------------------------------------------------------
    E_AXIS_STATE.AXIS_IDLE:
      _eResult                      := AxisCamIdle(TRUE);
  
    //---------------------------------------------------------------------------
    E_AXIS_STATE.CAM_IN:
      _eResult                      := AxisCamIn(TRUE);
  
    //--------------------------------------------------------------------------
    E_AXIS_STATE.CAM_OUT:
      _eResult                      := AxisCamOut(TRUE);
  
    //--------------------------------------------------------------------------
    E_AXIS_STATE.CAM_SCALING:
      _eResult                      := AxisCamScaling(TRUE);
  
    //--------------------------------------------------------------------------
    E_AXIS_STATE.CAM_INFO:
      _eResult                      := AxisCamInfo(TRUE);
  
    //--------------------------------------------------------------------------
    E_AXIS_STATE.CAM_RD_MOTION_FUNCTION:
      _eResult                      := AxisReadMotionFunction(TRUE);
  
    //--------------------------------------------------------------------------
    E_AXIS_STATE.CAM_RD_MOTION_FUNCTION_POINT:
      _eResult                      := AxisReadMotionFunctionPoint(TRUE);
  
    //--------------------------------------------------------------------------
    E_AXIS_STATE.CAM_WRT_MOTION_FUNCTION:
      _eResult                      := AxisWriteMotionFunction(TRUE);
  
    //--------------------------------------------------------------------------
    E_AXIS_STATE.CAM_WRT_MOTION_FUNCTION_POINT:
      _eResult                      := AxisWriteMotionFunctionPoint(TRUE);
  
  ELSE
    IF (_eCmd > E_AXIS_CTRL.AXIS_NULL)
    THEN
      _eResult                      := E_PROGRESS.PROGRESS_NOT_EXIST;
      _State^[_nAxisIndex].bError   := TRUE;
    ELSE
      _eResult                      := E_PROGRESS.PROGRESS_INVALID;
    END_IF
  END_CASE
END_CASE
//-----------------------------------------------------------------------------
//-----------------------------------------------------------------------------
//  OnChange of execution state result
//    - log result and clear error number on interface
//-----------------------------------------------------------------------------
IF (_eResult <> _eResultOld)
THEN
  LogResult();
  _eResultOld                       := _eResult;
END_IF
//-----------------------------------------------------------------------------
//-----------------------------------------------------------------------------
//  CAM couplingstate and TableId freom AXIS_REF
//-----------------------------------------------------------------------------
_State^[_nAxisIndex].wCamCouplingState   := CouplingState;
_State^[_nAxisIndex].nCamCouplingTableId := _AxisSlave.NcToPlc.CamCouplingTableID;
//-----------------------------------------------------------------------------
END_METHOD

PROPERTY ItfMcAxes : array[1..MAX_AXIS] of I_McAxis
SET
_ItfMcAxis := ItfMcAxes;
END_SET
END_PROPERTY

METHOD LogCheck
VAR_INST
  _sChck            : STRING(30);

  _stMsg            : ST_Message;
END_VAR
  _stMsg.eType               := SEL((_eCheck = E_CHECK_STATE.CHECK_DONE),(E_MessageType.eMessageError),(E_MessageType.eMessageInfo));
  _stMsg.eDevice             := E_Device.Camming + (_AxisSlave.NcToPlc.AxisId);
  _stMsg.eSubdevice          := e_Subdevice.CamControl;
  _stMsg.iErrorNumber        := _nAxisIndex;

  _sChck                     := concat('E_CHECK_STATE', '.');
  _sChck                     := concat(_sChck, TO_STRING(_eCheck));

  _stMsg.sText               := concat('cyclic check: ', _sChck);

  IF (_MessageLevel > E_MessageType.eMessageError)
  THEN
    f_MessageSet(_stMsg);
  ELSE
    IF (_stMsg.eType = E_MessageType.eMessageError)
    THEN
      f_MessageSet(_stMsg);
    END_IF
  END_IF
END_METHOD

METHOD PRIVATE LogControl
VAR_INST
  _sResult,
  _sCtrl            : STRING(30);

  _stMsg            : ST_Message;
END_VAR
  _stMsg.eType               := E_MessageType.eMessageInfo;
  _stMsg.eDevice             := E_Device.Camming + (_AxisSlave.NcToPlc.AxisId);
  _stMsg.eSubdevice          := e_Subdevice.CamControl;
  _stMsg.iErrorNumber        := _nAxisIndex;

  _sCtrl                     := concat('E_AXIS_CTRL', '.');
  _sCtrl                     := concat(_sCtrl, TO_STRING(_eCmd));

  _stMsg.sText               := concat('new command: ', _sCtrl);

  IF (_MessageLevel > E_MessageType.eMessageError)
  THEN
    f_MessageSet(_stMsg);
  ELSE
    IF (_stMsg.eType = E_MessageType.eMessageError)
    THEN
      f_MessageSet(_stMsg);
    END_IF
  END_IF
END_METHOD

METHOD PRIVATE LogResult
VAR_INST
  _sResult,
  _sCtrl            : STRING(30);

  _stMsg            : ST_Message;
END_VAR

  _stMsg.eType               := E_MessageType.eMessageInfo;
  _stMsg.eDevice             := E_Device.Camming + (_AxisSlave.NcToPlc.AxisId);
  _stMsg.eSubdevice          := e_Subdevice.CamControl;
  _stMsg.iErrorNumber        := _nAxisIndex;

  _sCtrl                     := concat('E_AXIS_CTRL', '.');
  _sCtrl                     := concat(_sCtrl, TO_STRING(_eCmdOld));

  _sResult                   := concat(': E_PROGRESS', '.');
  _sResult                   := concat(_sResult, TO_STRING(_eResult));

  _stMsg.sText               := concat(_sCtrl, ' ');
  _stMsg.sText               := concat(_sCtrl, _sResult);

  IF (_MessageLevel > E_MessageType.eMessageError)
  THEN
    f_MessageSet(_stMsg);
  ELSE
    IF (_stMsg.eType = E_MessageType.eMessageError)
    THEN
      f_MessageSet(_stMsg);
    END_IF
  END_IF
END_METHOD

PROPERTY MotionFunction : POINTER TO ARRAY[1..MAX_AXIS] OF ST_MOTION_FUNCTION
SET
_MotionFunction := MotionFunction;
END_SET
END_PROPERTY

PROPERTY MotionFunctionPoint : pointer to array[1..MAX_AXIS] of ST_MOTION_FUNCTION_POINT
SET
_MotionFunctionPoint := MotionFunctionPoint;
END_SET
END_PROPERTY

END_FUNCTION_BLOCK

// ---- CAM/FB_CamAxis.TcPOU
FUNCTION_BLOCK abstract FB_CamAxis
VAR
  _eCheck                       : E_CHECK_STATE;
  _nErrorId                     : UDINT; // datafield for error

  _MessageLevel                 : E_MessageType;

  _AxisSlave                    : REFERENCE TO AXIS_REF;
  _AxisMaster                   : REFERENCE TO AXIS_REF;

  _fbCamInV2                    : Tc2_MC2_Camming.MC_CamIn_V2;
  _fbScalingV2                  : Tc2_MC2_Camming.MC_CamScaling_V2;
  _fbCamInfoV2                  : Tc2_MC2_Camming.MC_CamInfo_V2;

  _fbCamOut                     : Tc2_MC2_Camming.MC_CamOut;

  _fbSetCamOnlineChangeMode     : Tc2_MC2_Camming.MC_SetCamOnlineChangeMode;

  _fbReadMotionFunction         : Tc2_MC2_Camming.MC_ReadMotionFunction;
  _fbReadMotionFunctionPoint    : Tc2_MC2_Camming.MC_ReadMotionFunctionPoint;
  _fbReadMotionFunctionValues   : Tc2_MC2_Camming.MC_ReadMotionFunctionValues;

  _fbWriteMotionFunction        : Tc2_MC2_Camming.MC_WriteMotionFunction;
  _fbWriteMotionFunctionPoint   : Tc2_MC2_Camming.MC_WriteMotionFunctionPoint;

  _stCamData                    : ST_CAM_DATA;  // camming parameters for function calls

  _mcCamInfoData                : Tc2_MC2_Camming.MC_CamInfoData; // read cam info from NC

  _mcCamRef                     : MC_CAM_REF;
  _mcMotionFunction             : ARRAY[1..MAX_MOTION_FUNCTION_POINTS] OF Tc2_MC2_Camming.MC_MotionFunctionPoint;
  _mcMotionFunctionPoint        : Tc2_MC2_Camming.MC_MotionFunctionPoint;
  _nMotionFunctionSize          : UINT;
END_VAR

METHOD CamIn : E_PROGRESS
VAR_INPUT
  Execute           : BOOL;
  nMasterIndex      : UINT;
END_VAR
VAR_INST
  _eCk              : E_CHECK_STATE;
  _eState           : E_PROGRESS;
  _rValue           : LREAL;
  _udiErr           : UDINT;
  _stMsg            : ST_Message;
END_VAR
IF NOT __ISVALIDREF(_AxisSlave)
THEN
  _eCheck                     := E_CHECK_STATE.CAM_SLAVE_AXIS_REF_INVALID;
  CamIn                       := E_PROGRESS.PROGRESS_ERROR;
  RETURN;
END_IF

IF NOT Execute THEN _eState := E_PROGRESS.PROGRESS_INIT; END_IF


CASE _eState
OF
  E_PROGRESS.PROGRESS_INIT:
    IF Execute 
    THEN
      memset(ADR(_stMsg),0,SIZEOF(_stMsg));
      _udiErr                       := 0;

      IF NOT (nMasterIndex = _stCamData.nMasterIndex)
      THEN
        _eState                     := E_PROGRESS.PROGRESS_ERROR;
        _eCk                        := E_CHECK_STATE.CAM_MASTER_AXIS_REF_INVALID;

        _stMsg.eType                := E_MessageType.eMessageError;
        _stMsg.eDevice              := E_Device.Camming + (_AxisSlave.NcToPlc.AxisId);
        _stMsg.eSubdevice           := e_Subdevice.fbCamInV2;
        _stMsg.iErrorNumber         := nMasterIndex;
  
        _stMsg.sText                := concat(' : ', TO_STRING(_eCk));
        f_MessageSet(_stMsg);

      ELSE
        _eState                     := E_PROGRESS.PROGRESS_BUSY;
        _eCk                        := E_CHECK_STATE.CHECK_DONE;

        IF (_MessageLevel = E_MessageType.eMessageVerbose)
        THEN
          _stMsg.eType              := E_MessageType.eMessageVerbose;
          _stMsg.eDevice            := E_Device.Camming + (_AxisSlave.NcToPlc.AxisId);
          _stMsg.eSubdevice         := e_Subdevice.fbCamInfoV2;
          _stMsg.iErrorNumber       := 0;
    
          _stMsg.sText              := concat(' : ', TO_STRING(_eState));
          f_MessageSet(_stMsg);
        END_IF

      _fbCamInV2(
          Master                    := _AxisMaster, 
          Slave                     := _AxisSlave, 
          Execute                   := FALSE, 
          ActivationMode            := _stCamData.nActivationMode, 
          ActivationPosition        := _stCamData.rActivationPosition, 
          CamTableID                := _stCamData.nCamTableId,
          Scaling                   := CamScalingData,
          Options                   := CamInOptions);
      END_IF
    END_IF
END_CASE
CASE _eState
OF
  E_PROGRESS.PROGRESS_BUSY:
    _fbCamInV2(
          Master                    := _AxisMaster, 
          Slave                     := _AxisSlave, 
          Execute                   := TRUE, 
          ActivationMode            := _stCamData.nActivationMode, 
          ActivationPosition        := _stCamData.rActivationPosition, 
          CamTableID                := _stCamData.nCamTableId);

    IF (_fbCamInV2.Error)
    THEN
      _eState                       := E_PROGRESS.PROGRESS_ERROR;
      _udiErr                       := _fbCamInV2.ErrorID;

      _stMsg.eType                  := E_MessageType.eMessageError;
      _stMsg.eDevice                := E_Device.Camming + (_AxisSlave.NcToPlc.AxisId);
      _stMsg.eSubdevice             := e_Subdevice.fbCamInV2;
      _stMsg.iErrorNumber           := _udiErr;

      _stMsg.sText                  := concat(' : ', TO_STRING(_eState));
      f_MessageSet(_stMsg);

      _fbCamInV2(
          Master                    := _AxisMaster, 
          Slave                     := _AxisSlave, 
          Execute                   := FALSE); 

    ELSIF (_fbCamInV2.InSync)
    THEN
      _eState                       := E_PROGRESS.PROGRESS_DONE;

      IF (_MessageLevel > E_MessageType.eMessageError)
      THEN
        _stMsg.eType                := E_MessageType.eMessageInfo;
        _stMsg.eDevice              := E_Device.Camming + (_AxisSlave.NcToPlc.AxisId);
        _stMsg.eSubdevice           := e_Subdevice.fbCamInV2;
        _stMsg.iErrorNumber         := 0;
  
        _stMsg.sText                := concat(' : ', TO_STRING(_eState));
        f_MessageSet(_stMsg);
      END_IF

